// height of the panel
g_panelHeight :LREAL := 0.009;

END_VAR

// ---- GVLs/SlaveArms/GVL_SlaveControlParameters.TcGVL
{attribute 'global_init_slot' := '49991'}
VAR_GLOBAL CONSTANT
	// slave arm joint position controller parameters
	g_posKp :ARRAY[1..g_sJntNum] OF LREAL :=[2000.0, 2000.0, 18000.0, 5(5)];
	g_posKd :ARRAY[1..g_sJntNum] OF LREAL :=[200.0, 200.0, 1800.0, 5(0.25)];
	g_posKi :ARRAY[1..g_sJntNum] OF LREAL :=[20000.0, 20000.0, 30000.0, 5(10.0)];
	g_posKiLimit :ARRAY[1..g_sJntNum] OF LREAL :=[2500,2500,  250, 5(75)];// define in current
	g_posCtrlLimit :ARRAY[1..g_sJntNum] OF LREAL :=[5600,5600,  500, 5(200)];// define in current
	
	// slave arm joint position controller parameters-----Modify joint stiffness---More flexible--1028
	g_allowLowStiff:BOOL:=FALSE;
	g_posKpLowStiff :ARRAY[1..g_sJntNum] OF LREAL :=[500.0, 500.0, 18000.0, 5(5)];
	g_posKdLowStiff :ARRAY[1..g_sJntNum] OF LREAL :=[200.0, 200.0, 1800.0, 5(0.25)];
	g_posKiLowStiff :ARRAY[1..g_sJntNum] OF LREAL :=[10000.0, 10000.0, 30000.0, 5(10.0)];
	g_posKiLimitLowStiff :ARRAY[1..g_sJntNum] OF LREAL :=[500,1000,  250, 5(75)];// define in current
	g_posCtrlLimitLowStiff :ARRAY[1..g_sJntNum] OF LREAL :=[500,1000,  500, 5(250)];// define in current
	
	// control tolerance
	g_jntCtrlAngTolLow :LREAL :=0.2*g_deg2Rad;
	g_jntCtrlAngTolHigh :LREAL :=2*g_deg2Rad;
	g_cartCtrlPosTolLow :LREAL :=0.0002;
	g_cartCtrlOriTolLow :LREAL :=0.2*g_deg2Rad;
	g_cartCtrlPosTolHigh :LREAL :=0.001;
	g_cartCtrlOriTolHigh :LREAL :=2*g_deg2Rad;
	
	// filter cut-off frequency for velocity and torque
	g_curJntVelLpfCutoffFreq :LREAL := 30;
	g_cmdJntTrqLpfCutoffFreq :LREAL := 300;
	g_curJntTrqLpfCutoffFreq :LREAL := 300;
		
	// controller would keep command unchanged when error 
	// between command and current value is less than this value
	g_jntCtrlErrForCmdHold :LREAL :=1.0*g_deg2Rad;
	
	// joint is assumed to be static if velocity is less than this value
	g_jntStaticVelThres :LREAL :=0.2*g_deg2Rad;
	
	// joint velocity threshold for full friction compensation
	g_fullFrictionVel :LREAL :=2.0*g_deg2Rad;
	
	// friciton compensation scael
	g_frictionCompScale :LREAL := 0.8;
	
END_VAR

// ---- GVLs/SlaveArms/GVL_SlaveJointEncoderCaliData.TcGVL
{attribute 'qualified_only'}
// Robot3 --joints parameters of slave arms
VAR_GLOBAL CONSTANT	
	// absolute encoder value at minimal joint positon
	g_minLinkEncoder :ARRAY[1..g_sArmNum, 1..g_sJntNum] OF DINT :=
		[796618, 12395160, 5368016, 0, 0, 0, 0, 0,
		 13317378, 3888760, 9175760, 0, 0, 0, 0, 0,
		 823964, 3955316, 15205696, 0, 0, 0, 0, 0,
		 4820816, 7977020, 9226720, 0, 0, 0, 0, 0];
		 
	// absolute encoder value at maximum joint positon
	g_maxLinkEncoder :ARRAY[1..g_sArmNum, 1..g_sJntNum] OF DINT :=
		[15464922, 5123844, 14570432, 0, 0, 0, 0, 0,
		 11230582, 13464106, 1613344, 0, 0, 0, 0, 0,
		 15526052, 13536910, 7701984, 0, 0, 0, 0, 0,
		 2731020, 789080, 1671808, 0, 0, 0, 0, 0];
	
	// absolute encoder value at calibrated positon
	g_caliLinkEncoder :ARRAY[1..g_sArmNum, 1..g_sJntNum] OF DINT :=
		[8162412, 8169482, 14570432, 15377856,15482848, 7058832, 7015248, 7155184,
		 3932766, 16656494, 1613344, 15324752, 15485488, 7135776, 7032592, 6946704,
		 8248074, 16595424, 7701984, 15349408, 15361392, 7017904, 6757296, 7028608,
		 12196142, 3807946, 1671808, 15274368, 15387696, 6812992, 7016768, 7073088];
	
	 // if absolute encoder value cross zeros within joint motion range
	 // NOTICE: joint 7 is always 0.
	g_linkEncZeroCross :ARRAY[1..g_sArmNum, 1..g_sJntNum] OF INT :=
		[0, 0, 0, 1, 1, 1, 1, 1,
		 1, 1, 1, 1, 1, 1, 1, 1,
		 0, 1, 1, 1, 1, 1, 1, 1,
		 1, 0, 1, 1, 1, 1, 1, 1];
		 
	 // joint SDO address
	g_slaveArmNetID: ARRAY[1..4] OF T_AmsNetId:=['169.254.186.39.3.1','169.254.186.39.8.1','169.254.186.39.9.1','169.254.186.39.10.1'];
	g_slaveJointNetPort:ARRAY[1..g_sArmNum,1..g_sJntNum] OF UINT :=[
		1006,	1007,	1008,	2(1009),	3(1010),
		1006,	1007,	1008,	2(1009),	3(1010),
		1006,	1007,	1008,	2(1009),	3(1010),
		1006,	1007,	1008,	2(1009),	3(1010)];
	g_slaveLEDNetPort:ARRAY[1..g_sArmNum] OF UINT :=[4(1004)];
		
//################ DO NOT modify parameters below ###########################
	// abolute encoder expanded limit buffer in case there is calibrtion error at limit position
	g_linkEncLimitBuffer : DINT := 100000;
	
	// absolute encoder direction
	g_asbEncoderDir :ARRAY[1..g_sJntNum] OF INT :=[1, -1, 1, 1, 1, 1, 1, 1];
	
	// flag if joint can rotate multiple cycles
	g_multipleCyclesJoint :ARRAY[1..g_sArmNum, 1..g_sJntNum] OF INT :=
		[0, 0, 0, 1, 1, 1, 1, 1,
		 0, 0, 0, 1, 1, 1, 1, 1,
		 0, 0, 0, 1, 1, 1, 1, 1,
		 0, 0, 0, 1, 1, 1, 1, 1];
		 
	// joint position at link encoder calibrated point
	g_linkEncCaliJntPos :ARRAY[1..g_sJntNum] OF LREAL :=[0.0, -PI/2 + 8*g_deg2rad, 0.581633, 5(0.0)];

	
END_VAR

// ---- GVLs/SlaveArms/GVL_SlaveMotorParameters.TcGVL
{attribute 'global_init_slot' := '49991'}
{attribute 'qualified_only'}
VAR_GLOBAL CONSTANT
	// encoder resolution
	g_incEncoderRes :ARRAY[1..g_sJntNum] OF DINT :=[8(65536)];
	g_absEncoderRes :ARRAY[1..g_sJntNum] OF DINT :=[8(16777216)];
	
	// reduction ratio
	g_motorReduction :ARRAY[1..g_sJntNum] OF LREAL :=[ 81,81,  (66.0/10)*2*pi/0.010, 5(388125.0/4693)];
	g_absEncoderReduction :ARRAY[1..g_sJntNum] OF LREAL :=[2(1.0), 2*PI/0.64, 5(1.0)];
	
	// motor parameters
	g_motorTrqConst :ARRAY[1..g_sJntNum] OF LREAL :=[ 0.16,0.16, 0.017,5(0.0193)];
	g_motorMaxCurrent :ARRAY[1..g_sJntNum] OF LREAL :=[ 5600,5600,  600, 5(250)];//mA
	
	// motor encoder direction
	g_motorDir :ARRAY[1..g_sJntNum] OF INT :=[-1, 1, -1, 1, 1, 1, 1, 1];
																 
	// joint position limit
	g_minJntPos: ARRAY[1..g_sJntNum] OF LREAL:=[-2.7,	-1.5-pi/2,	0.23, 	5(-g_largeNum)];	
	g_maxJntPos: ARRAY[1..g_sJntNum] OF LREAL:=[2.7,	1.13-pi/2, 	0.58, 		5(g_largeNum)];
	
	// DH joint position limit
	//NOTE: wrist pitch and yaw angle is reset after instrument is mounted 
	g_minDHJntPos : ARRAY[1..6] OF LREAL :=[-2.7,	-1.2-pi/2,	0.235, -5.5, -PI/2 - 75*g_deg2Rad , -PI/2];
	g_maxDHJntPos : ARRAY[1..6] OF LREAL :=[2.7,	1-pi/2, 	0.575, 5.5, -PI/2 + 75*g_deg2Rad, PI/2];
	
	// joint velocity limit
	g_maxJntVel :ARRAY[1..g_sJntNum] OF LREAL :=[1.25, 1.25, 0.25, 5(7.0)];
		
END_VAR

// ---- FBs_CartControlles/I_CartJointCtrl.TcIO
INTERFACE I_CartJointCtrl

METHOD init : BOOL
VAR_IN_OUT CONSTANT
	i_slaveCart	:FB_SlaveCart;
END_VAR
VAR_IN_OUT 
	r_cartCtrlCmd :ST_SlaveArmCtrlCmds;
END_VAR
END_METHOD

PROPERTY isFinished : BOOL
GET
END_GET
END_PROPERTY

METHOD reset : BOOL
VAR_INPUT
END_VAR
END_METHOD

METHOD run : BOOL
VAR_IN_OUT CONSTANT
	i_slaveCart	:FB_SlaveCart;
END_VAR
VAR_IN_OUT 
	r_cartCtrlCmd :ST_SlaveArmCtrlCmds;
END_VAR
END_METHOD

END_INTERFACE

// ---- FBs_SlaveControllers/I_SlaveArmCtrl.TcIO
INTERFACE I_SlaveArmCtrl

METHOD init : BOOL
VAR_IN_OUT CONSTANT
	i_slaveArm	:FB_SlaveArm;
END_VAR
VAR_IN_OUT 
	r_slaveArmCtrlCmd :ST_SlaveArmCtrlCmds;
END_VAR
END_METHOD

PROPERTY isFinished : bool
GET
END_GET
END_PROPERTY

METHOD reset : BOOL
VAR_INPUT
END_VAR
END_METHOD

METHOD run : BOOL

VAR_IN_OUT CONSTANT
	i_endoscopePose : ST_Frame;
	i_masterStatus :ST_MasterStatus;
	i_setupStatus: ST_SetupStatus;
	i_slaveArm :FB_SlaveArm;
	
END_VAR
VAR_IN_OUT
	r_slaveArmCtrlCmd :ST_SlaveArmCtrlCmds;
END_VAR
END_METHOD

PROPERTY timePeriod : lreal
GET
END_GET
END_PROPERTY

END_INTERFACE

// ---- Mains/CartControl.TcPOU
PROGRAM CartControl
VAR
	// cart instance
	m_cartRobot :FB_CartRobot;
	
	// Output cart status
	m_cartStatus AT%Q* : ST_CartStatus;
	
	// cart joint data
	m_cartJointsData AT %Q* :ST_CartJointData;
	
	m_cartDataPool: ST_CartInputDataPool;
	
	// wait time before cart init for ethercat to be statble 
	m_cartInitWaitTime : LREAL:=0;
	
	// cart init flag
	m_cartInit :BOOL :=FALSE;
	
	m_workHeartTon0 : TON;
	m_workHeartTon1 : TON;
	
	m_cartInSterileStateTon :Ton;
	m_cartInSterileState :BOOL;
	//Aseptic sleeve is installed flag
	m_asepticInstalledFlag : Vec4b;
	m_slaveArmDisableFlag : Vec4b;
END_VAR

// wait communication to be stable
IF(m_cartInitWaitTime<g_robotInitWaitTime) THEN
	m_cartInitWaitTime := m_cartInitWaitTime+g_cartCtrlCycleTime;
	RETURN;
END_IF

// cart init
IF m_cartInit =FALSE THEN
	m_cartRobot.Init();
	m_cartInit:=TRUE;
END_IF

// input from UI
UIInputProcess();

// cart run
m_cartRobot.run(m_cartDataPool);

m_cartRobot.getStatus(m_cartStatus,m_cartJointsData);


UIOutputProcess();

// tranform data from UI(global variable write by ADS) to ST_UIData
METHOD UIInputProcess : BOOL
VAR_INPUT
END_VAR
VAR
	i:int;
END_VAR
// cart Joystick data
m_cartDataPool.m_UIData.m_joystickDataFromUI := GVL_interactUI.g_joystickSignalArray;

m_cartDataPool.m_UIData.m_ctrlEnableFromUI := GVL_interactUI.g_uiCtrl;

//limit_height:UINT;  上位机的高度值单位是mm，系统的高度值单位是m，底座高度是1805mm
//打开ui_control.limit_height_adjusting后可以调整立柱，并实时将立柱当前高度上传
IF (GVL_interactUI.g_uiCtrl.m_heightLimitAdjustEnable=TRUE) THEN
	m_cartDataPool.m_UIData.m_standColumnHightLimit := GVL_CartMotorParameters.g_maxJntPos[5];
ELSIF  (GVL_interactUI.g_uiCtrl.m_heightLimitAdjustEnable=FALSE) AND GVL_interactUI.g_heightLimitEnbale AND ABS((m_cartDataPool.m_UIData.m_standColumnHightLimit *1000+1850)-GVL_interactUI.g_heightLimitFromUI)>5 THEN
	m_cartDataPool.m_UIData.m_standColumnHightLimit := UINT_TO_LREAL(GVL_interactUI.g_heightLimitFromUI-GVL_CartControlParameters.g_cartInitialHeight)/1000;
ELSIF GVL_interactUI.g_heightLimitEnbale=FALSE THEN
	m_cartDataPool.m_UIData.m_standColumnHightLimit := GVL_CartMotorParameters.g_maxJntPos[5];
END_IF
GVL_interactUI.g_heightLimit :=LREAL_TO_UINT (m_cartRobot.m_slaveCart.curJntPos[5] * 1000 + GVL_CartControlParameters.g_cartInitialHeight);

//Surgical orientation selection
m_cartDataPool.m_UIData.m_surgicalSite := GVL_interactUI.g_surgicalSite;
m_cartDataPool.m_UIData.m_surgicalLocation := GVL_interactUI.g_surgicalLocation;
END_METHOD

METHOD UIOutputProcess : BOOL
VAR_INPUT
END_VAR
VAR 
	i : INT;
END_VAR
//TODO
//work heart
m_workHeartTon0(IN:= GVL_interactUI.g_heartBeat = 1, PT:= T#1S, Q=> , ET=> );
m_workHeartTon1(IN:= GVL_interactUI.g_heartBeat = 0, PT:= T#1S, Q=> , ET=> );
IF m_workHeartTon0.Q THEN
	GVL_interactUI.g_heartBeat :=0 ;
ELSIF m_workHeartTon1.Q THEN
	GVL_interactUI.g_heartBeat  :=1 ;
END_IF

GVL_interactUI.g_cartOperation.m_drapingAdjustState := m_cartRobot.m_slaveCart.m_cartDataFromUI.m_cartDrapingState;
GVL_interactUI.g_cartOperation.m_dockingAdjustState := m_cartRobot.m_slaveCart.m_cartDataFromUI.m_cartDockingState;

GVL_interactUI.g_trocarStatus := INT_TO_BOOL(m_cartRobot.m_slaveCart.m_trocarOnFlag);

GVL_interactUI.g_slaveRunAlone := NOT SlaveArmControl.m_slaveRobot.m_masterOnLine;
GVL_interactUI.g_joysticksTrigger := SafetyCheck.m_joysticksTrigger;

IF GVL_interactUI.g_surgicalStatus = 1 THEN
	IF NOT SlaveArmControl.m_slaveRobotData.m_asepticDeployCompletedFlag THEN
		m_slaveArmDisableFlag := g_zeroVec4b;
	END_IF
	GVL_interactUI.g_cartOperation.m_setupSterileState := BOOL_TO_UINT(m_asepticInstalledFlag[1]) OR BOOL_TO_UINT(m_asepticInstalledFlag[2]) OR BOOL_TO_UINT(m_asepticInstalledFlag[3]) OR BOOL_TO_UINT(m_asepticInstalledFlag[4]) ;
ELSE
	GVL_interactUI.g_cartOperation.m_setupSterileState := BOOL_TO_UINT(m_asepticInstalledFlag[1]) AND BOOL_TO_UINT(m_asepticInstalledFlag[2]) AND BOOL_TO_UINT(m_asepticInstalledFlag[3]) AND BOOL_TO_UINT(m_asepticInstalledFlag[4]) ;
	m_slaveArmDisableFlag := SlaveArmControl.m_slaveInputDataPool.m_UIData.m_slaveArmDisableFlag;	
	Gvl_interactUI.g_InstruSeriesRecord := g_zeroInstruRecord;
END_IF

FOR i := 1 TO 4 BY 1 DO
	m_asepticInstalledFlag[i] := m_slaveArmDisableFlag[i] OR SlaveArmControl.m_slaveRobot.m_panelMountedFlag[i];
END_FOR

GVL_interactUI.g_cartOperation.m_setupSterileStateArm1 := BOOL_TO_UINT(m_asepticInstalledFlag[1]); 
GVL_interactUI.g_cartOperation.m_setupSterileStateArm2 := BOOL_TO_UINT(m_asepticInstalledFlag[2]); 
GVL_interactUI.g_cartOperation.m_setupSterileStateArm3 := BOOL_TO_UINT(m_asepticInstalledFlag[3]); 
GVL_interactUI.g_cartOperation.m_setupSterileStateArm4 := BOOL_TO_UINT(m_asepticInstalledFlag[4]); 

GVL_interactUI.g_cartOperation.m_scopeInstalled := BOOL_TO_UINT(m_cartDataPool.m_slaveStatus.m_endoscopeMounted);

FOR i := 1 TO 4 BY 1 DO
	IF SlaveArmControl.m_slaveRobot.m_slaveArms[i].instrument.Instrutype<>InstruType_endoscope THEN
		IF SlaveArmControl.m_slaveRobot.m_instrumentMountedFlag[i] AND SlaveArmControl.m_slaveRobot.m_endoscopeMounted AND GVL_interactUI.g_cartOperation.m_setupSterileState = 1 THEN
			GVL_interactUI.g_cartOperation.m_inSurgicalAllowed := 1;
			EXIT;
		ELSE
			GVL_interactUI.g_cartOperation.m_inSurgicalAllowed := 0;
		END_IF	
	END_IF	
END_FOR


//Cart_static_in_sterile_state:UINT; //台车进入无菌区，并且台车停止运动(连续10s没有运动)，0：没有完成，1：完成
IF m_cartRobot.m_slaveCart.m_cartDataFromUI.m_cartDockingState = 1 THEN
	IF m_cartRobot.m_CartState = CartJointState_Movement THEN
		m_cartInSterileState := FALSE;
	ELSIF m_cartRobot.m_lastCartState = CartJointState_Movement THEN
		m_cartInSterileState := TRUE;
	END_IF
ELSE
	m_cartInSterileState := FALSE;
	GVL_interactUI.g_cartOperation.m_cartInSterileState:=0;
END_IF
m_cartInSterileStateTon(IN:= m_cartInSterileState, PT:= T#10S, Q=> , ET=> );
IF m_cartInSterileStateTon.Q THEN
	GVL_interactUI.g_cartOperation.m_cartInSterileState:=1;
END_IF
END_METHOD

END_PROGRAM

// ---- FBs_Robots/FB_CartRobot.TcPOU
FUNCTION_BLOCK FB_CartRobot
VAR_INPUT
END_VAR
VAR_OUTPUT
END_VAR
VAR

	m_slaveCart: FB_SlaveCart;		
	
	// input arm button 
	m_carHandChassisDriveUnlock AT%I* :ARRAY [1..2] OF BOOL;
	
	//open laser io
	m_openHorizonLaser AT  %Q* :DINT;
	m_openCrossLaser AT  %Q* :DINT;

	m_joystickData:Vec8d;

	// all cart controller instance 
	m_cartCtrlFactory :ARRAY[1..CartJointState_totalNum] OF I_CartJointCtrl;
	
	m_cartState:E_CartJointState:=CartJointState_Init;
	m_lastCartState:E_CartJointState:=CartJointState_Init;
	m_nextCartState:E_CartJointState:=CartJointState_Init;
	
	// flag if cart joint self-check passed
	m_selfCheckPass:  BOOL :=FALSE;
	
	// all cart controller instance 
	m_cartError :FB_CartCtrlError;
	m_cartInit :FB_CartCtrlInit;
	m_cartReady :FB_CartCtrlReady;
	m_cartInSurgery :FB_CartCtrlInSurgery;
	m_cartMotionCar :FB_CartCtrlMotionCar;
	m_cartAsepticDeploy :FB_CartCtrlAsepticDeploy;
	m_cartAdjust :FB_CartCtrlAdjust;
	m_cartRotaOverhang :FB_CartCtrlRotaOverhang;
	m_cartSlowStop : FB_CartCtrlSlowDown;
	m_cartStandColuAdjust : FB_CartCtrlStandColuAdjust;
	
	// cart controller interface
	m_cartCtrl : I_CartJointCtrl;
	m_cartCtrlCmds : ST_SlaveArmCtrlCmds;
	
	//state machine flow jump condition allowed
	m_hangAdjustAllowed : BOOL;
	m_asepticDeploymentAllowed :BOOL;
	m_cartMoveAllowed :BOOL;
	m_rotaOverhangAllowed :BOOL;
END_VAR

METHOD getStatus : BOOL
VAR_IN_OUT
	
	r_cartStatus :ST_CartStatus;	

	// cart joint data
	r_cartJointsData :ST_CartJointData;
END_VAR

VAR 
	i : INT;
END_VAR
r_cartStatus.m_CartState :=m_cartState;

r_cartStatus.m_uiControl := GVL_interactUI.g_uiCtrl;
r_cartStatus.m_cartDumpEnergy := GVL_interactUI.g_dumpEnergyUPS;
r_cartStatus.m_sdrivingLeverSensorManualFlag :=NOT m_slaveCart.m_drivingLeverSensorManual;
//r_cartStatus.m_stabilizerDeployedFlag
r_cartStatus.m_trocarOnFlag := m_slaveCart.m_trocarOnFlag;
r_cartStatus.m_joystickValue := m_slaveCart.m_joystickSignal;
r_cartStatus.m_jntPosReachLimit := m_cartAdjust.jntPosReachLimit;

r_cartJointsData.m_cmdJntPos := m_slaveCart.cmdJntPos;
r_cartJointsData.m_cmdJntVel := m_slaveCart.cmdJntVel;
r_cartJointsData.m_curJntPos := m_slaveCart.curJntPos;
r_cartJointsData.m_curJntTrq := m_slaveCart.curJntCurrent;
r_cartJointsData.m_curJntVel := m_slaveCart.curJntVel;
r_cartJointsData.m_curLinkPos := m_slaveCart.curLinkPos;
r_cartJointsData.m_curMotorPos := m_slaveCart.curMotorPos;
END_METHOD

METHOD init : BOOL
VAR_INPUT
END_VAR
VAR
	i:INT;
END_VAR

m_slaveCart.init();
m_cartState := CartJointState_Init;
m_lastCartState := CartJointState_Init;
m_nextCartState := CartJointState_Init;
m_selfCheckPass := FALSE;

//command init
m_cartCtrlCmds.m_jntEnableFlag := g_zeroVec8i;
m_cartCtrlCmds.m_jntOPMode := g_slaveAllPosMode;
m_cartCtrlCmds.m_cmdJntPos := m_slaveCart.m_curJntPos;
m_cartCtrlCmds.m_cmdJntVel := g_zeroVec8d;
m_cartCtrlCmds.m_cmdJntAcc := g_zeroVec8d;
m_cartCtrlCmds.m_cmdJntTrq := g_zeroVec8d;


// generate controller factory
//m_cartCtrlFactory[CartJointState_Error] := m_cartError;
m_cartCtrlFactory[CartJointState_Init] := m_cartInit;
m_cartCtrlFactory[CartJointState_Ready] := m_cartReady;
m_cartCtrlFactory[CartJointState_InSurgery] := m_cartInSurgery;
m_cartCtrlFactory[CartJointState_Movement] := m_cartMotionCar;
m_cartCtrlFactory[CartJointState_HangAdjust] := m_cartAdjust;
m_cartCtrlFactory[CartJointState_AsepticDeployment] := m_cartAsepticDeploy;
m_cartCtrlFactory[CartJointState_RotaOverhang] := m_cartRotaOverhang;
m_cartCtrlFactory[CartJointState_SlowStop] := m_cartSlowStop;
m_cartCtrlFactory[CartJointState_StandColuAdjust] := m_cartStandColuAdjust;

// assign controller
m_cartCtrl:=m_cartCtrlFactory[m_cartState];
m_cartCtrl.Init(m_slaveCart,m_cartCtrlCmds);
END_METHOD

METHOD laserIO : BOOL
VAR_INPUT
END_VAR

//cross laser IO output , when slave self check succeed , and trocar  install at least one
IF GVL_interactUI.g_slaveSelfCheckStatus = 2 AND m_slaveCart.m_trocarOnFlag = 0 THEN
	m_openCrossLaser := 1;
ELSE
	m_openCrossLaser := 0;
END_IF

//Horizontal laser IO output ,when adjusting the trolley or moving the trolley
IF (m_slaveCart.curJntPos[5] * 1000 + GVL_CartControlParameters.g_cartInitialHeight) > GVL_CartControlParameters.g_cartOpenHorizonLaserHeight AND  (m_cartState = CartJointState_Movement OR m_cartState = CartJointState_HangAdjust) THEN
	m_openHorizonLaser :=  1;
ELSE
	m_openHorizonLaser :=  0;
END_IF
END_METHOD

METHOD PUBLIC run : BOOL
VAR_IN_OUT CONSTANT
	i_cartDataPool: ST_CartInputDataPool;
END_VAR
VAR
	i:INT;
END_VAR
// state machine transition
stateMachine(i_cartDataPool);	

//update ui data
m_slaveCart.ProcessingUIData(i_cartDataPool.m_UIData);

//update cart joint status
m_slaveCart.updateStatus();

laserIO();

// null ptr check
IF 0 = m_cartCtrl THEN
	RETURN;
END_IF

// run controller
m_cartCtrl.run(m_slaveCart,m_cartCtrlCmds);


m_slaveCart.updateCmds(m_cartCtrlCmds);
END_METHOD

METHOD PROTECTED stateMachine : BOOL
VAR_IN_OUT CONSTANT
	i_cartDataPool: ST_CartInputDataPool;
END_VAR
VAR
	i,j:INT;
END_VAR
m_hangAdjustAllowed := m_slaveCart.m_trocarOnFlag=0 AND ( i_cartDataPool.m_UIData.m_ctrlEnableFromUI.m_joystickEnable OR i_cartDataPool.m_UIData.m_ctrlEnableFromUI.m_cameraJoystickEnable);
m_asepticDeploymentAllowed := m_slaveCart.m_trocarOnFlag=0 AND ((i_cartDataPool.m_UIData.m_ctrlEnableFromUI.m_dockingEnable AND m_slaveCart.cartDockingState=0) 
												OR (i_cartDataPool.m_UIData.m_ctrlEnableFromUI.m_drapingEnable AND m_slaveCart.cartDrapingState=0)) AND NOT ( i_cartDataPool.m_safetyData.m_cartAdjustErr OR i_cartDataPool.m_safetyData.m_cartStandColumnErr) ;
m_cartMoveAllowed := m_slaveCart.m_trocarOnFlag=0 AND  m_carHandChassisDriveUnlock[1] AND m_carHandChassisDriveUnlock[2] AND NOT i_cartDataPool.m_safetyData.m_cartWheelErr;
m_rotaOverhangAllowed := m_slaveCart.m_trocarOnFlag=0 AND m_slaveCart.m_rotaOverhangOnFlag > 0 AND NOT i_cartDataPool.m_safetyData.m_cartOverhangErr;

// state machine transit
CASE m_cartState OF
	//cart joint error
	CartJointState_Error:
		//IF FALSE = i_cartDataPool.m_safetyData.m_slaveErrFlag THEN
		//	// to standby
		//	IF m_selfCheckPass THEN
		//		m_nextCartState :=CartJointState_Standby;
		//	ELSE
		//		m_nextCartState :=CartJointState_Init;
		//	END_IF
		//END_IF

	CartJointState_Init:
		IF m_cartCtrl.isFinished THEN
			m_nextCartState :=CartJointState_Ready;
		END_IF
		
		
	CartJointState_Ready:
		IF m_cartCtrl.isFinished  THEN
			m_nextCartState := CartJointState_InSurgery;
			
		ELSIF m_hangAdjustAllowed THEN
			m_nextCartState := CartJointState_HangAdjust;
			
		ELSIF m_asepticDeploymentAllowed THEN
			m_nextCartState := CartJointState_AsepticDeployment;
			
		ELSIF m_cartMoveAllowed THEN
			m_nextCartState := CartJointState_Movement;
			
		ELSIF m_rotaOverhangAllowed THEN
			m_nextCartState := CartJointState_RotaOverhang;
			
		ELSIF m_slaveCart.m_trocarOnFlag=0 AND  m_slaveCart.m_columnAdjustEnable  THEN
			m_nextCartState := CartJointState_StandColuAdjust;
		END_IF
		
	
	CartJointState_InSurgery:
		IF m_cartCtrl.isFinished  THEN
			m_nextCartState :=CartJointState_Ready;
		END_IF
		
		
	CartJointState_Movement:
		IF m_slaveCart.m_trocarOnFlag<>0 OR (NOT m_carHandChassisDriveUnlock[1] AND NOT m_carHandChassisDriveUnlock[2])  THEN
			m_nextCartState :=CartJointState_Ready;
		ELSIF i_cartDataPool.m_safetyData.m_cartWheelErr THEN
			m_nextCartState :=CartJointState_Ready;
		END_IF
		
		
	CartJointState_HangAdjust:
		IF  m_slaveCart.m_trocarOnFlag<>0 OR (NOT i_cartDataPool.m_UIData.m_ctrlEnableFromUI.m_joystickEnable AND NOT i_cartDataPool.m_UIData.m_ctrlEnableFromUI.m_cameraJoystickEnable ) THEN
			m_nextCartState :=CartJointState_SlowStop;
		END_IF
		
		
	CartJointState_AsepticDeployment:
		IF m_cartCtrl.isFinished  THEN
			IF i_cartDataPool.m_UIData.m_ctrlEnableFromUI.m_dockingEnable THEN
				m_slaveCart.cartDockingState := 1;
			ELSIF i_cartDataPool.m_UIData.m_ctrlEnableFromUI.m_drapingEnable THEN
				m_slaveCart.cartDrapingState := 1;
			END_IF
			m_nextCartState :=CartJointState_SlowStop;
		ELSIF i_cartDataPool.m_safetyData.m_cartAdjustErr OR i_cartDataPool.m_safetyData.m_cartStandColumnErr THEN
			m_nextCartState :=CartJointState_Ready;
		ELSIF m_slaveCart.m_trocarOnFlag<>0 OR (NOT i_cartDataPool.m_UIData.m_ctrlEnableFromUI.m_dockingEnable AND NOT i_cartDataPool.m_UIData.m_ctrlEnableFromUI.m_drapingEnable) THEN
			m_nextCartState :=CartJointState_SlowStop;
		END_IF
		
		
	CartJointState_RotaOverhang:
		IF m_slaveCart.m_rotaOverhangOnFlag = 0 OR  m_slaveCart.m_trocarOnFlag<>0  THEN
			m_nextCartState :=CartJointState_SlowStop;
		ELSIF i_cartDataPool.m_safetyData.m_cartOverhangErr THEN
			m_nextCartState :=CartJointState_Ready;
		END_IF
		
	CartJointState_StandColuAdjust:
		IF (m_slaveCart.m_trocarOnFlag<>0 OR i_cartDataPool.m_safetyData.m_cartStandColumnErr) OR  NOT m_slaveCart.m_columnAdjustEnable  THEN
			m_nextCartState :=CartJointState_SlowStop;
		END_IF	
	
	CartJointState_SlowStop:
		IF m_cartCtrl.isFinished  THEN
			m_nextCartState :=CartJointState_Ready;
		END_IF
END_CASE

// Controller transit
IF m_nextCartState<> m_cartState THEN
	//reset current controller
	m_cartCtrl.reset();
	
	// transit to new controller
	m_lastCartState:=m_cartState;
	m_cartState:=m_nextCartState;
	m_cartCtrl:=m_cartCtrlFactory[m_cartState];
	
	//init next controller
	m_cartCtrl.Init(m_slaveCart, m_cartCtrlCmds);
	m_slaveCart.updateCmds(m_cartCtrlCmds);
END_IF
END_METHOD

END_FUNCTION_BLOCK

// ---- FBs_Robots/FB_SlaveCart.TcPOU
FUNCTION_BLOCK FB_SlaveCart
VAR
	
	//Driving force of the car io
	m_driveForce AT %I* :Vec2i;
	
	//stabilizing foot sensor  (normally-closed contact)
	m_stabilizFootSensorLeft AT%I* :BOOL;
	m_stabilizFootSensorRight AT%I* :BOOL;
	m_drivingLeverSensorAuto AT%I* :BOOL;
	m_drivingLeverSensorManual AT%I* :BOOL;
	
	//Trocar IO check
	m_trocarIO AT %I* : ARRAY [1..4] OF UDINT;
	m_trocarCheck : ARRAY [1..4] OF FB_trocarDetect;
	m_trocarFlag : ARRAY [1..4] OF BOOL;
	m_trocarOnFlag : INT:=0;
	
	//output screw break IO 
	m_screwBreak AT %Q* : BOOL;
	m_screwBreakSR : SR;
	
	//car overhang rotation signal is in the arm
	m_carRotaOverhangIO AT%I* : ARRAY [1..4] OF UDINT;
	m_rotaButtonDetect : ARRAY [1..4] OF FB_rotaButtonDetect;
	m_rotaOverhangOnFlag : UDINT :=0;
	
	//cart joint
	m_cartJoints: ARRAY [1..g_cartJntNum] OF FB_CartJoint;
	
	// cart status
	m_cartStatus  : ST_CartStatus;
	
	//cart joint 5 enable detect
	m_standColumnEnableDetect : FB_cartJntEnableDetect;
	m_standColumnDisenableDetect : FB_cartJntDisenableDetect;

	// arm joint data
	m_curMotorPos :Vec8d;
	m_curLinkPos :Vec8d;
	m_curLinkSingle :Vec8d;
	m_curJntPos :Vec8d;
	m_curDHJntPos :Vec6d;
	m_curGripAngle :LREAL;
	m_curJntVel :Vec8d;
	m_curDHJntVel :Vec6d;
	m_curJntTrq :Vec8d;
	m_rawJntCurrent :Vec8d;
	m_filtJntCurrent :Vec8d;
	m_cmdJntTrq :Vec8d;
	m_cmdJntCurrent : Vec8d;
	m_cmdJntPos :Vec8d;
	m_cmdJntVel :Vec8d;

	//SDO Writer
	m_CommunicationCycleInitMZSub1:ARRAY [1..3] OF FB_EcCoESdoWrite;
	m_CommunicationCycleInitMZSub2:ARRAY [1..3] OF FB_EcCoESdoWrite;
	m_CommunicationCycleSub1:INT:=1;
	m_CommunicationCycleSub2:INT:=-3;
	
	//update ui information
	m_joystickSignal:Vec8d;
	m_cartDataFromUI : ST_CartUIData;
	m_ctrlEnable : ST_uiControl;
	m_surgicalStatusF : F_TRIG;
	
	//stand column adjust of setup joint 3
	m_columnJntVel : LREAL;
	m_columnAdjustEnable : BOOL;
	m_limitBufferForCtrl : LREAL := 0.01;
	m_midJntPos : LREAL := 0.1;
	enableTon : ARRAY [1..4] OF FB_TON;
	
	// collision detection
	m_collisionDetection : FB_CartCollisionDetect;
	m_collisionFlag :BOOL:=false;
END_VAR

PROPERTY cartDockingState : UINT
GET
END_GET
SET
m_cartDataFromUI.m_cartDockingState := cartDockingState;
END_SET
END_PROPERTY

PROPERTY cartDrapingState : UINT
GET
END_GET
SET
m_cartDataFromUI.m_cartDrapingState := cartDrapingState;
END_SET
END_PROPERTY

METHOD checkIO : BOOL
VAR_INPUT
END_VAR
VAR
	i:INT;
END_VAR
//check overhang rotation button
m_rotaOverhangOnFlag := MAX( m_rotaButtonDetect[1].run(m_carRotaOverhangIO[1]), m_rotaButtonDetect[2].run(m_carRotaOverhangIO[2]),m_rotaButtonDetect[3].run(m_carRotaOverhangIO[3]),m_rotaButtonDetect[4].run(m_carRotaOverhangIO[4]));

FOR i := 1 TO g_sArmNum BY 1 DO
	//trocar in place monitor
	m_trocarFlag[i] := m_trocarCheck[i].run(m_trocarIO[i] );
END_FOR

m_trocarOnFlag := BOOL_TO_INT(m_trocarFlag[1]) + BOOL_TO_INT(m_trocarFlag[2]) + BOOL_TO_INT(m_trocarFlag[3]) + BOOL_TO_INT(m_trocarFlag[4]);

//setup robot joint 3 adjust and drive column movement
m_columnAdjustEnable :=columnAdjustEnable(o_columnJntVel => m_columnJntVel  );
END_METHOD

PROPERTY cmdJntPos : REFERENCE TO Vec8d
GET
cmdJntPos REF= m_cmdJntPos;
END_GET
END_PROPERTY

PROPERTY cmdJntVel : REFERENCE TO Vec8d
GET
cmdJntVel REF= m_cmdJntVel;
END_GET
END_PROPERTY

METHOD columnAdjustEnable : BOOL
VAR_INPUT
END_VAR

VAR_OUTPUT
	o_columnJntVel : LREAL;
END_VAR

VAR_STAT
	curJntPos : vec4d;
	curJntVel : vec4d;
	columnJntVel : vec4d;
	adjustStartFlag : vec4b;
	m_columnAdjustEnable : vec4b;
END_VAR
VAR
	i : INT;
	armId : INT;
	limitDis : vec4d;
	m_adjustFlag : vec4b;
END_VAR

FOR i := 1 TO g_sArmNum DO
	curJntPos[i] := SetupArmControl.m_setupRobot.m_setupArms[i].m_curJntPos[3];
	curJntVel[i] := SetupArmControl.m_setupRobot.m_setupArms[i].m_curJntVel[3];
	m_adjustFlag[i] := SetupArmControl.m_setupRobot.m_setupArms[i].m_manualAdjustOnFlag AND m_trocarOnFlag=0 AND SetupArmControl.m_setupRobot.m_setupArmState[i] = SetupArmState_ManualAdjust 
									AND NOT SafetyCheck.m_SafetyCheck.m_jntErrFlag[i,0,2] AND NOT SafetyCheck.m_SafetyCheck.m_jntErrFlag[i,0,3] AND NOT SafetyCheck.m_SafetyCheck.m_jntErrFlag[i,3,3] AND NOT SafetyCheck.m_SafetyCheck.m_jntErrFlag[i,2,3] ;
	
	IF m_adjustFlag[i] THEN
		limitDis[i] := MIN(GVL_SetupMotorParameters.g_maxJntPos[i,3] - curJntPos[i], curJntPos[i]-GVL_SetupMotorParameters.g_minJntPos[i,3]);
		IF limitDis[i] < m_limitBufferForCtrl THEN
			adjustStartFlag[i] := TRUE; 
			columnJntVel[i] := sign(m_midJntPos - curJntPos[i]) * GVL_CartControlParameters.g_maxJntVel[5];
		
		ELSIF limitDis[i] >= m_limitBufferForCtrl AND NOT m_columnAdjustEnable[i] THEN
			columnJntVel[i] := 0;
			adjustStartFlag[i] := FALSE;
			
		ELSE
			IF curJntVel[i] <> 0 AND adjustStartFlag[i] THEN
				columnJntVel[i] := -LIMIT(-GVL_CartControlParameters.g_maxJntVel[5], curJntVel[i], GVL_CartControlParameters.g_maxJntVel[5]);
			END_IF
		END_IF
		
		armId := i;
		enableTon[i](IN:= adjustStartFlag[i], PT:= T#3S, Q=> m_columnAdjustEnable[i], ET=> );
		EXIT;
	ELSE
		adjustStartFlag[i] := FALSE;
		columnJntVel[i] := 0;
	END_IF
	enableTon[i](IN:= adjustStartFlag[i], PT:= T#3S, Q=> m_columnAdjustEnable[i], ET=> );
END_FOR

//output stand column joint velocity and start adjust single
IF armId > 0 THEN
	o_columnJntVel := columnJntVel[armId];
END_IF
columnAdjustEnable := m_columnAdjustEnable[1] OR m_columnAdjustEnable[2] OR m_columnAdjustEnable[3] OR m_columnAdjustEnable[4];
END_METHOD

PROPERTY ctrlEnable : REFERENCE TO ST_uiControl
GET
ctrlEnable REF= m_ctrlEnable;
END_GET
SET
END_SET
END_PROPERTY

PROPERTY curDHJntPos :REFERENCE TO Vec6d
GET
curDHJntPos ref= m_curDHJntPos;
END_GET
END_PROPERTY

PROPERTY curDHJntVel :REFERENCE TO Vec6d
GET
curDHJntVel REF= m_curDHJntVel;
END_GET
END_PROPERTY

PROPERTY curJntCurrent :REFERENCE TO Vec8d
GET
curJntCurrent ref=m_filtJntCurrent;
END_GET
END_PROPERTY

PROPERTY curJntPos : REFERENCE TO Vec8d
GET
curJntPos ref=m_curJntPos;
END_GET
END_PROPERTY

PROPERTY curJntVel :REFERENCE TO Vec8d
GET
curJntVel ref=m_curJntVel;
END_GET
END_PROPERTY

PROPERTY curLinkPos :REFERENCE TO Vec8d
GET
curLinkPos ref=m_curLinkPos;
END_GET
END_PROPERTY

PROPERTY curMotorPos : REFERENCE TO  Vec8d
GET
curMotorPos ref=m_curMotorPos;
END_GET
END_PROPERTY

METHOD PUBLIC enable : BOOL
VAR_IN_OUT CONSTANT
	i_jntIdx :Vec8i;
END_VAR
VAR
	i :INT ;
END_VAR
FOR i:=1 TO g_cartJntNum DO
	IF 3<=i AND i<5 THEN
		IF 1= i_jntIdx[i] THEN
			m_cartJoints[i].enableMZ();
		ELSE
			m_cartJoints[i].disable();
		END_IF
	ELSIF i = 5 THEN
		IF 1= i_jntIdx[i] THEN
			m_screwBreak := m_standColumnEnableDetect.run(IOValue:= m_cartJoints[i].enableMZ());
			m_standColumnDisenableDetect.run(IOValue:=FALSE );
		ELSE
			m_standColumnEnableDetect.run(IOValue:= FALSE);
			m_screwBreak :=  NOT m_standColumnDisenableDetect.run(IOValue:=m_cartJoints[i].disable());
		END_IF
	ELSE
		IF 1= i_jntIdx[i] THEN
			m_cartJoints[i].enable();
		ELSE
			m_cartJoints[i].disable();
		END_IF
	END_IF
END_FOR
END_METHOD

METHOD init : BOOL
VAR_INPUT
END_VAR
VAR
	i:INT;
END_VAR


// cart joint init
FOR i:= 1 TO g_cartJntNum BY 1 DO
	m_cartJoints[i].init(i, g_cartCtrlCycleTime);
END_FOR


// joint init
FOR i:=1 TO g_cartJntNum DO
	m_cartJoints[i].initJntPos();
END_FOR


// update cart status if joint position is re-init
updateStatus();



//MingZhi drive example Initialize the communication period
FOR i := 1 TO 3 BY 1 DO
	m_CommunicationCycleInitMZSub1[i](sNetID:= GVL_CartJointEncoderCaliData.g_slaveCartNetID,
				nSlaveAddr := GVL_CartJointEncoderCaliData.g_slaveCartJointNetPort[i+2],
				nSubIndex:=1,nIndex:=16#60C2,pSrcBuf:=ADR(m_CommunicationCycleSub1),cbBufLen:=SIZEOF(m_CommunicationCycleSub1),bExecute:=TRUE);
	
	IF NOT m_CommunicationCycleInitMZSub1[i].bBusy THEN
		m_CommunicationCycleInitMZSub1[i](bExecute:=FALSE);
	END_IF
					
	m_CommunicationCycleInitMZSub2[i](sNetID:= GVL_CartJointEncoderCaliData.g_slaveCartNetID,
					nSlaveAddr := GVL_CartJointEncoderCaliData.g_slaveCartJointNetPort[i+2],
					nSubIndex:=2,nIndex:=16#60C2,pSrcBuf:=ADR(m_CommunicationCycleSub2),cbBufLen:=SIZEOF(m_CommunicationCycleSub2),bExecute:=TRUE);
	
	IF NOT m_CommunicationCycleInitMZSub2[i].bBusy THEN
		m_CommunicationCycleInitMZSub2[i](bExecute:=FALSE);
	END_IF
END_FOR
END_METHOD

METHOD  joystickSignalAnalysis : Vec8d 
VAR_INPUT
	i_joystickDataFromUI:ARRAY [0..21] OF USINT;
END_VAR

VAR_STAT
	i:INT;
	m_handData:ARRAY [0..21] OF USINT;
	m_outHandData : Vec8d;
END_VAR

IF i_joystickDataFromUI[0] = 16#FF THEN
	m_handData := i_joystickDataFromUI;
	m_outHandData[1] :=m_handData[7]*256 + m_handData[8]; // car  joint5 pillar
	m_outHandData[2] :=m_handData[3]*256 + m_handData[4]; //car joint7 beamStretch
	m_outHandData[3] :=m_handData[1]*256 + m_handData[2]; // car joint6  beamRot
	m_outHandData[4] :=m_handData[5]*256 + m_handData[6]; // joint8 overhang 
	m_outHandData[5] :=m_handData[9]*256 + m_handData[10];
	m_outHandData[6] :=m_handData[11]*256 + m_handData[12];
	m_outHandData[7] :=m_handData[13]*256 + m_handData[14];
	m_outHandData[8] :=m_handData[15]*256 + m_handData[16];
END_IF
joystickSignalAnalysis:=m_outHandData;
END_METHOD

METHOD ProcessingUIData : BOOL
VAR_IN_OUT CONSTANT
	//UI information, import from UI controller
	i_UIData :ST_CartUIData;
END_VAR
VAR
	i : INT;
END_VAR
m_joystickSignal := joystickSignalAnalysis(i_UIData.m_joystickDataFromUI);

m_ctrlEnable:=i_UIData.m_ctrlEnableFromUI;

m_cartDataFromUI.m_standColumnHightLimit := i_UIData.m_standColumnHightLimit;

m_cartDataFromUI.m_cartSpecificPosDraping := GVL_CartControlParameters.g_surgicalDrapingPos;

FOR i := 1 TO g_sArmNum BY 1 DO
	IF i_UIData.m_surgicalSite > 0 AND i_UIData.m_surgicalLocation > 0 THEN
		m_cartDataFromUI.m_cartSpecificPosDocking[i + 4] := GVL_CartControlParameters.g_surgicalOrientPos[i_UIData.m_surgicalSite, i_UIData.m_surgicalLocation,i];
	END_IF
END_FOR

m_surgicalStatusF(CLK:= GVL_interactUI.g_surgicalStatus , Q=> );
IF m_surgicalStatusF.Q THEN
	cartDrapingState := 0;
END_IF

IF NOT (m_cartDataFromUI.m_surgicalSite = i_UIData.m_surgicalSite) OR NOT (m_cartDataFromUI.m_surgicalLocation = i_UIData.m_surgicalLocation) THEN
	cartDockingState := 0;
END_IF

m_cartDataFromUI.m_surgicalSite := i_UIData.m_surgicalSite;
m_cartDataFromUI.m_surgicalLocation := i_UIData.m_surgicalLocation;
END_METHOD

PROPERTY status : ST_CartStatus
GET
status := m_cartStatus;
END_GET
END_PROPERTY

METHOD PUBLIC updateCmds : BOOL
VAR_IN_OUT CONSTANT
	i_cartCtrlCmd : ST_SlaveArmCtrlCmds;
END_VAR
VAR
	i:INT;
END_VAR
m_cmdJntTrq:=i_cartCtrlCmd.m_cmdJntTrq;
m_cmdJntPos :=i_cartCtrlCmd.m_cmdJntPos;
m_cmdJntVel :=i_cartCtrlCmd.m_cmdJntVel;


// enable/disable joints
enable(i_cartCtrlCmd.m_jntEnableFlag);

// position/Velocity control
FOR i:=1 TO g_sJntNum DO 
	IF i_cartCtrlCmd.m_jntOPMode[i]=DriverOPMode_Pos THEN
		m_cmdJntTrq[i]:=0;
		m_cmdJntVel[i]:=0;
		m_cartJoints[i].updateCmd(DriverOPMode_Pos,m_cmdJntPos[i],m_cmdJntTrq[i],m_cmdJntVel[i]);
	ELSIF i_cartCtrlCmd.m_jntOPMode[i]=DriverOPMode_Vel THEN
		m_cmdJntTrq[i]:=0;
		m_cmdJntPos[i]:=0;
		m_cartJoints[i].updateCmd(DriverOPMode_Pos,m_cmdJntPos[i],m_cmdJntTrq[i],m_cmdJntVel[i]);
	ELSIF i_cartCtrlCmd.m_jntOPMode[i]=DriverOPMode_MZPos  THEN
		m_cmdJntTrq[i]:=0;
		m_cmdJntVel[i]:=0;
		//Input torque mode because the operating mode word for the contour position mode of the MingZhi driver is 1
		m_cartJoints[i].updateCmd(DriverOPMode_Trq,m_cmdJntPos[i],m_cmdJntTrq[i],m_cmdJntVel[i]);
	ELSIF i_cartCtrlCmd.m_jntOPMode[i]=DriverOPMode_cspMZ  THEN
		 m_cartJoints[i].updateCmd(DriverOPMode_cspMZ,m_cmdJntPos[i],m_cmdJntTrq[i],m_cmdJntVel[i]);
	ELSIF DriverOPMode_csvMZ = i_cartCtrlCmd.m_jntOPMode[i] THEN
		m_cartJoints[i].updateCmd(DriverOPMode_csvMZ,m_cmdJntPos[i],m_cmdJntTrq[i],m_cmdJntVel[i]);
	END_IF
END_FOR

// collision check
m_collisionFlag := m_collisionDetection.run(m_rawJntCurrent, m_cmdJntPos, m_curJntVel);
END_METHOD

METHOD PUBLIC updateStatus : BOOL
VAR_INPUT
END_VAR
VAR
	i:INT;
END_VAR
// update joint data
FOR i:=1 TO g_sJntNum DO
	m_cartJoints[i].updateStatus();
END_FOR

//IO output   Horizontal laser IO output   Cross laser IO output
checkIO();


// get joint data
FOR i:=1 TO g_cartJntNum DO
	m_curMotorPos[i]:=m_cartJoints[i].motorPos;
	m_curLinkPos[i]:=m_cartJoints[i].linkPos;
	m_curLinkSingle[i]:=m_cartJoints[i].linkSingle;
	m_curJntPos[i]:=m_cartJoints[i].jntPos;
	m_curJntVel[i]:=m_cartJoints[i].jntVel;
	m_curJntTrq[i]:=m_cartJoints[i].jntTrq;
	m_rawJntCurrent[i]:=m_cartJoints[i].rawCurrent;
	m_filtJntCurrent[i]:=m_cartJoints[i].filtCurrent;
	m_cmdJntCurrent[i]:=m_cartJoints[i].cmdCurrent;
END_FOR
END_METHOD

END_FUNCTION_BLOCK

// ---- FBs_Auxiliary/FB_trocarDetect.TcPOU
FUNCTION_BLOCK FB_trocarDetect
VAR_INPUT
END_VAR
VAR_OUTPUT
END_VAR
VAR
	m_trocarOnCounts :INT :=0;
	m_trocarOnCountThres :INT :=50;
END_VAR

// check if instrument is on
METHOD run : BOOL
VAR_INPUT
	IOValue :UDINT;
END_VAR
// trocar io is 5th bit 
IF 32=(IOValue AND 10#32) THEN
	m_trocarOnCounts :=MIN(m_trocarOnCounts +1,m_trocarOnCountThres);
ELSE
	m_trocarOnCounts :=0;
END_IF

run := m_trocarOnCounts >= m_trocarOnCountThres;
END_METHOD

END_FUNCTION_BLOCK

// ---- FBs_Auxiliary/FB_rotaButtonDetect.TcPOU
FUNCTION_BLOCK FB_rotaButtonDetect
VAR_INPUT
END_VAR
VAR_OUTPUT
END_VAR
VAR
	m_rotaButtonUpOnCounts :INT :=0;
	m_rotaButtonUpOnCountThres :INT :=50;
	m_rotaButtonDownOnCounts :INT :=0;
	m_rotaButtonDownOnCountThres :INT :=-50;
END_VAR

// check if instrument is on
METHOD run : UDINT
VAR_INPUT
	IOValue :UDINT;
END_VAR
// 
IF 1=(IOValue AND 16#01) OR 2=(IOValue AND 16#02) THEN
	m_rotaButtonUpOnCounts :=MIN(m_rotaButtonUpOnCounts +1,m_rotaButtonUpOnCountThres);
ELSE
	m_rotaButtonUpOnCounts :=0;
END_IF

IF m_rotaButtonUpOnCounts >= m_rotaButtonUpOnCountThres THEN
	run := IOValue;
ELSE
	run := 0;
END_IF
END_METHOD

END_FUNCTION_BLOCK

// ---- FBs_Robots/FB_CartJoint.TcPOU
FUNCTION_BLOCK FB_CartJoint EXTENDS FB_JointBase
VAR_INPUT
END_VAR
VAR_OUTPUT
END_VAR
VAR
	//Cart motor output IO
	m_cartMotorOutput AT %Q*	:ST_CartMotorOutput;
	
	m_cmdAcc:LREAL;
	
END_VAR

METHOD cmd2motorMZ : DINT
VAR_INPUT
	i_cmd:LREAL;
	i_controlCycleTime :LREAL;
END_VAR
cmd2motorMZ:=LREAL_TO_DINT(((4*m_motorEncoderRes*m_motorReduction*i_controlCycleTime)/(2*pi))*i_cmd*65536);
END_METHOD

METHOD PUBLIC enableMZ : BOOL
VAR_INPUT
END_VAR
IF (MZDriverStatusWord_SwitchOnDisable AND m_motorInputs.m_statusWord) = MZDriverStatusWord_SwitchOnDisable    THEN
	m_motorOutputs.m_controlWord:=DriverCtrlWord_INIT;
	enableMZ := FALSE;
ELSIF (MZDriverStatusWord_OperationEnbale AND m_motorInputs.m_statusWord) = MZDriverStatusWord_OperationEnbale THEN
	enableMZ :=  TRUE;
ELSIF (MZDriverStatusWord_SwitchOn AND m_motorInputs.m_statusWord) =  MZDriverStatusWord_SwitchOn THEN
	m_motorOutputs.m_controlWord:=DriverCtrlWord_OP;
	enableMZ :=  FALSE;
ELSIF (MZDriverStatusWord_ReadyToSwitchOn AND m_motorInputs.m_statusWord) = MZDriverStatusWord_ReadyToSwitchOn THEN
	m_motorOutputs.m_controlWord:=DriverCtrlWord_PREOP;
	enableMZ :=  FALSE;
ELSIF (MZDriverStatusWord_Fault AND m_motorInputs.m_statusWord) = MZDriverStatusWord_Fault THEN
	m_motorOutputs.m_controlWord:=DriverCtrlWord_FaultReset;
//ELSE
//	m_motorOutputs.m_controlWord:=DriverCtrlWord_INIT;
//	enable :=  FALSE;
END_IF
END_METHOD

METHOD PUBLIC init : BOOL
VAR_INPUT
	i_jntIdx :INT;
	i_controlCycleTime :LREAL;
END_VAR
m_jntIdx:=i_jntIdx;
m_cycleTime := i_controlCycleTime;

// hardware parameters
m_motorEncoderRes :=GVL_CartMotorParameters.g_incEncoderRes[i_jntIdx];
m_linkEncoderRes :=GVL_CartMotorParameters.g_absEncoderRes[i_jntIdx];
m_motorReduction :=GVL_CartMotorParameters.g_motorReduction[i_jntIdx];
m_linkEncoderReduction :=GVL_CartMotorParameters.g_absEncoderReduction[i_jntIdx];
m_trqConst :=GVL_CartMotorParameters.g_motorTrqConst[i_jntIdx];
m_maxCurrent :=GVL_CartMotorParameters.g_motorMaxCurrent[i_jntIdx];
m_motorDir :=GVL_CartMotorParameters.g_motorDir[i_jntIdx];								
m_minJntPos	:=GVL_CartMotorParameters.g_minJntPos[i_jntIdx];
m_maxJntPos	:=GVL_CartMotorParameters.g_maxJntPos[i_jntIdx];

//link encoder calibartion data
m_linkEncoderDir :=GVL_CartJointEncoderCaliData.g_asbEncoderDir[i_jntIdx];
m_minLinkEncoder :=GVL_CartJointEncoderCaliData.g_minLinkEncoder[ i_jntIdx] - m_linkEncoderDir*GVL_SetupJointEncoderCaliData.g_linkEncLimitBuffer; // expand limit
m_maxLinkEncoder :=GVL_CartJointEncoderCaliData.g_maxLinkEncoder[ i_jntIdx] + m_linkEncoderDir*GVL_SetupJointEncoderCaliData.g_linkEncLimitBuffer; // expand limit
m_caliLinkEncoder :=GVL_CartJointEncoderCaliData.g_caliLinkEncoder[ i_jntIdx];
m_linkEncCaliJntPos :=GVL_CartJointEncoderCaliData.g_linkEncCaliJntPos[i_jntIdx];
m_linkEncZeroCross :=GVL_CartJointEncoderCaliData.g_linkEncZeroCross[ i_jntIdx];
m_multiCycles :=GVL_CartJointEncoderCaliData.g_multipleCyclesJoint[i_jntIdx];

// convert cali link encoder if joint cross zero
IF 1=m_linkEncZeroCross THEN
	IF 1=m_linkEncoderDir AND m_caliLinkEncoder < m_minLinkEncoder THEN
		m_caliLinkEncoder := GVL_CartJointEncoderCaliData.g_caliLinkEncoder[ i_jntIdx] + m_linkEncoderRes;
	ELSIF -1=m_linkEncoderDir AND m_caliLinkEncoder < m_maxLinkEncoder THEN
		m_caliLinkEncoder := GVL_CartJointEncoderCaliData.g_caliLinkEncoder[ i_jntIdx] + m_linkEncoderRes;
	END_IF
END_IF

// macro data
m_trq2CurrentRatio:=m_motorDir * 1000.0/(m_trqConst*m_motorReduction);
m_current2TrqRatio:=m_motorDir * (m_trqConst*m_motorReduction)/1000.0;
m_linkEnc2PosRatio := 2*PI*m_linkEncoderDir/(m_linkEncoderReduction*m_linkEncoderRes);
m_motorEnc2PosRatio := 2*PI * m_motorDir/(m_motorReduction * m_motorEncoderRes);


// motor data init
m_rawJntVel :=0;
m_curJntVel:=0;
m_curJntTrq :=0;
m_rawCurrent :=0;
m_filtCurrent :=0;
m_cmdJntVel :=0.0;
m_cmdJntTrq :=0.0;
m_cmdCurrent := 0.0;

// filter init
m_jntVelLpf.init(1, GVL_CartControlParameters.g_curJntVelLpfCutoffFreq, g_cartCtrlFreq);
m_cmdTrqLpf.init(1, GVL_CartControlParameters.g_cmdJntTrqLpfCutoffFreq, g_cartCtrlFreq);
m_curTrqLpf.init(1, GVL_CartControlParameters.g_curJntTrqLpfCutoffFreq, g_cartCtrlFreq);

// driver init value
m_motorOutputs.m_controlWord:=DriverCtrlWord_INIT;
m_motorOutputs.m_opMode:=INT_TO_SINT(DriverOPMode_Pos);
m_motorOutputs.m_cmdCurrent:=0;
m_motorOutputs.m_cmdMotorEncoder:=m_motorInputs.m_motorEncoder;
END_METHOD

METHOD PUBLIC updateCmd : BOOL
VAR_INPUT
	i_opMode : E_DriverOPMode;
	i_cmdPos :LREAL;
	i_cmdTrq :LREAL;
	i_cmdVel :LREAL;
END_VAR
VAR
	i:INT;
END_VAR
m_motorOutputs.m_opMode:=INT_TO_SINT( i_opMode);

// pos mode
IF i_opMode = DriverOPMode_Pos OR i_opMode = DriverOPMode_cspMZ  THEN
	m_motorOutputs.m_cmdCurrent:=0;
	m_cmdJntPos :=i_cmdPos;
	m_motorOutputs.m_cmdMotorEncoder :=motorPos2Enc(m_cmdJntPos);
ELSIF i_opMode = DriverOPMode_Vel THEN
	m_cmdJntVel := i_cmdVel;
	m_cartMotorOutput.m_cmdVelMzVelMode := cmd2motorMZ(m_cmdJntVel, g_cartCtrlCycleTime);
ELSIF i_opMode = DriverOPMode_Trq THEN   //Here the torque mode is equal to the contour position mode of the MingZhi driver
	m_cmdJntVel := i_cmdVel;
	m_cmdAcc:=i_cmdVel*2;
	m_cmdJntPos:=i_cmdPos;
	m_cartMotorOutput.m_cmdAccMz :=cmd2motorMZ(m_cmdAcc, g_cartCtrlCycleTime);
	m_cartMotorOutput.m_cmdVelMz := cmd2motorMZ(m_cmdJntVel, g_cartCtrlCycleTime);
	m_motorOutputs.m_cmdMotorEncoder := motorPos2Enc(m_cmdJntVel);
ELSIF i_opMode = DriverOPMode_csvMZ THEN
	m_cmdJntVel := i_cmdVel;
	m_cartMotorOutput.m_cmdVelMzVelMode := cmd2motorMZ(m_cmdJntVel, g_cartCtrlCycleTime);
END_IF
END_METHOD

METHOD PUBLIC updateStatus : BOOL
VAR_INPUT
END_VAR
// compute joint position
m_curLinkPos:= linkEnc2Pos();
m_curMotorPos:=motorEnc2Pos();
m_curLinkSingle := m_curLinkPos - 2*PI* m_linkEncCycles;

// Cart joint1-4 have no link enconder, use motor position
IF m_jntIdx <= 4 THEN
	m_curJntPos := m_curMotorPos;
ELSE
	m_curJntPos := m_curLinkPos;
END_IF

// compute joint velocity
m_curVelCalCycles := m_curVelCalCycles+1;
IF m_curVelCalCycles > m_velCalcCycles THEN
	m_rawJntVel:= (m_curJntPos-m_lastJntPos)/(m_cycleTime*m_velCalcCycles);
	m_curJntVel := m_jntVelLpf.run(m_rawJntVel);
	m_lastJntPos :=m_curJntPos;	
	m_curVelCalCycles:=1;
END_IF


// current and torque
m_rawCurrent := m_motorInputs.m_current;
m_filtCurrent := m_curTrqLpf.run(m_rawCurrent);
m_curJntTrq := m_filtCurrent * m_current2TrqRatio;
END_METHOD

END_FUNCTION_BLOCK

// ---- FBs_Robots/FB_JointBase.TcPOU
FUNCTION_BLOCK FB_JointBase
VAR_INPUT
END_VAR
VAR_OUTPUT
END_VAR
VAR
	// arm and joint index
	m_armIdx :INT;
	m_jntIdx :INT;
	
	// motor IO
	m_motorInputs AT%I*	:ST_MotorInputs;
	m_motorOutputs AT%Q* :ST_MotorOutputs;
	
	// cycle time
	m_cycleTime :LREAL;
	
	// calibrated link encoder data
	m_minLinkEncoder :DINT;
	m_maxLinkEncoder :DINT;
	m_caliLinkEncoder :DINT;
	m_linkEncCaliJntPos :LREAL;
	m_linkEncZeroCross :INT;
	m_initMotorEnc : DINT;
	m_multiCycles :INT;
	
	// joint position from link encoder after power on
	m_initLinkPos :LREAL;
	
	// data for link encoder multiple cycles
	m_lastLinkEncoder :DINT;
	m_linkEncCycles:INT;
	
	// device paramters
	m_motorEncoderRes :DINT;
	m_linkEncoderRes :DINT;
	m_motorReduction :LREAL;
	m_linkEncoderReduction :LREAL;
	m_trqConst :LREAL;
	m_maxCurrent :LREAL;
	m_motorDir :INT;								
	m_linkEncoderDir :INT;
	m_minJntPos: LREAL;
	m_maxJntPos: LREAL;
	
	// macro defined data for quick calculation
	m_trq2CurrentRatio:LREAL;
	m_current2TrqRatio:LREAL;
	m_linkEnc2PosRatio :LREAL;
	m_motorEnc2PosRatio :LREAL;
	
	// joint data
	m_curMotorPos :LREAL;
	m_curLinkPos :LREAL;
	m_curLinkSingle :LREAL;//[0-360]
	m_curJntPos	:LREAL;
	m_curJntVel :LREAL;
	m_rawJntVel :LREAL;
	m_curJntTrq :	LREAL;
	m_rawCurrent : LREAL;
	m_filtCurrent : LREAL;
	m_cmdJntPos :LREAL;
	m_cmdJntVel :LREAL;
	m_cmdJntTrq :LREAL;
	m_cmdCurrent : LREAL;
	m_lastJntPos :LREAL;
	
	// velocity filter
	m_jntVelLpf :FB_LowPassFilter;
	
	// command torque filter
	m_curTrqLpf : FB_LowPassFilter;
	m_cmdTrqLpf :FB_LowPassFilter;
	
	// velocity is calculated every (m_velCalcCycles) control cycles
	// TODO: insturment joint motor can not reach 4k now, so calculate their velocity with 1k frequency, need to remove later
	m_velCalcCycles :INT :=1;
	m_curVelCalCycles :INT :=1;
	
	// SDO writer
	m_opModeSDOWrite:FB_EcCoESdoWrite;
	m_MotorCurrentSDOWrite:FB_EcCoESdoWrite;
	
END_VAR

PROPERTY cmdCurrent : LREAL
GET
cmdCurrent:=m_cmdCurrent;
END_GET
END_PROPERTY

METHOD PUBLIC disable : BOOL
VAR_INPUT
END_VAR
m_motorOutputs.m_controlWord:=DriverCtrlWord_INIT;
disable:=true;
END_METHOD

PROPERTY driveInput : ST_MotorInputs
GET
driveInput := m_motorInputs;
END_GET
END_PROPERTY

PROPERTY driveOutput : ST_MotorOutputs
GET
driveOutput := m_motorOutputs;
END_GET
END_PROPERTY

METHOD PUBLIC enable : BOOL
VAR_INPUT
END_VAR
IF DriverStatusWord_INIT = m_motorInputs.m_statusWord THEN
	m_motorOutputs.m_controlWord:=DriverCtrlWord_PREOP;
	enable := FALSE;
ELSIF DriverStatusWord_PREOP = m_motorInputs.m_statusWord THEN
	m_motorOutputs.m_controlWord:=DriverCtrlWord_OP;
	enable :=  FALSE;
ELSIF DriverStatusWord_OP = m_motorInputs.m_statusWord THEN
	enable :=  TRUE;
//ELSE
//	m_motorOutputs.m_controlWord:=DriverCtrlWord_INIT;
//	enable :=  FALSE;
END_IF
END_METHOD

PROPERTY filtCurrent : LREAL
GET
filtCurrent:=m_filtCurrent;
END_GET
END_PROPERTY

METHOD PUBLIC initJntPos : BOOL
VAR_INPUT
END_VAR
m_lastLinkEncoder :=m_motorInputs.m_linkEncoder;
m_linkEncCycles:=0;
m_curLinkPos :=linkEnc2Pos();
m_initLinkPos:=m_curLinkPos;
m_initMotorEnc :=m_motorInputs.m_motorEncoder;
m_curMotorPos:=motorEnc2Pos();
m_curJntPos := m_curMotorPos;
m_cmdJntPos :=m_curJntPos;	
m_lastJntPos :=m_curJntPos;
END_METHOD

PROPERTY initLinkPos : lreal
GET
initLinkPos:=m_initLinkPos;
END_GET
SET
m_initLinkPos:=initLinkPos;
END_SET
END_PROPERTY

METHOD PUBLIC isEnabled : BOOL
VAR_INPUT
END_VAR
isEnabled :=(DriverStatusWord_OP = m_motorInputs.m_statusWord);
END_METHOD

PROPERTY jntPos : LREAL
GET
jntPos := m_curJntPos;
END_GET
END_PROPERTY

PROPERTY jntTrq : LREAL
GET
jntTrq:=m_curJntTrq;
END_GET
END_PROPERTY

PROPERTY jntVel : LREAL
GET
jntVel := m_curJntVel;
END_GET
END_PROPERTY

METHOD PROTECTED linkEnc2Pos : LREAL
VAR_INPUT
END_VAR
VAR
	incLinkPos :LREAL;
	newLinkEnc :DINT;
END_VAR
// cycle check
IF 1=m_multiCycles THEN
	IF (m_motorInputs.m_linkEncoder - m_lastLinkEncoder)*m_linkEncoderDir < -m_linkEncoderRes/2 THEN
		m_linkEncCycles :=m_linkEncCycles+1;
	ELSIF (m_motorInputs.m_linkEncoder - m_lastLinkEncoder)*m_linkEncoderDir > m_linkEncoderRes/2 THEN
		m_linkEncCycles :=m_linkEncCycles-1;
	END_IF
END_IF
m_lastLinkEncoder:=m_motorInputs.m_linkEncoder;

// convert link encoder if joint cross zero
newLinkEnc := m_motorInputs.m_linkEncoder;
IF 1=m_linkEncZeroCross AND 0 = m_multiCycles THEN
	IF 1=m_linkEncoderDir AND m_motorInputs.m_linkEncoder < m_minLinkEncoder THEN
		newLinkEnc := m_motorInputs.m_linkEncoder + m_linkEncoderRes;
	ELSIF -1=m_linkEncoderDir AND m_motorInputs.m_linkEncoder < m_maxLinkEncoder THEN
		newLinkEnc := m_motorInputs.m_linkEncoder + m_linkEncoderRes;
	END_IF
END_IF

// motion from calibrated points
incLinkPos := (newLinkEnc-m_caliLinkEncoder)*m_linkEnc2PosRatio;

// absolute joint position
linkEnc2Pos := incLinkPos + m_linkEncCaliJntPos + 2*PI* m_linkEncCycles;
END_METHOD

PROPERTY PUBLIC linkPos : LREAL
GET
linkPos:=m_curLinkPos;
END_GET
END_PROPERTY

PROPERTY linkSingle : LREAL
GET
linkSingle :=m_curLinkSingle;
END_GET
END_PROPERTY

METHOD PROTECTED motorEnc2Pos : LREAL
VAR_INPUT
END_VAR
motorEnc2Pos:= (m_motorInputs.m_motorEncoder-m_initMotorEnc)* m_motorEnc2PosRatio +m_initLinkPos;
END_METHOD

PROPERTY PUBLIC motorPos : LREAL
GET
motorPos := m_curMotorPos;
END_GET
END_PROPERTY

METHOD PROTECTED motorPos2Enc : DINT
VAR_INPUT
	i_jntPos :LREAL;
END_VAR

VAR
END_VAR
motorPos2Enc := LREAL_TO_DINT((i_jntPos-m_initLinkPos)/m_motorEnc2PosRatio + m_initMotorEnc);
END_METHOD

PROPERTY rawCurrent : LREAL
GET
rawCurrent := m_rawCurrent;
END_GET
END_PROPERTY

METHOD PROTECTED singleCyclePos : LREal
VAR_INPUT
END_VAR
VAR
	cycles :lreal;
END_VAR
cycles := ABS(FLOOR( m_curJntPos/g_2pi));
IF m_curJntPos<0 THEN
	singleCyclePos := m_curJntPos+cycles*g_2pi;
ELSE
	singleCyclePos := m_curJntPos-cycles*g_2pi;
END_IF
END_METHOD

METHOD PUBLIC updateCmds : BOOL
VAR_INPUT
	i_opMode : E_DriverOPMode;
	i_cmdPos :LREAL;
	i_cmdTrq :LREAL;
END_VAR
VAR
	filtCmdTrq :LREAL;
END_VAR
m_motorOutputs.m_opMode:=INT_TO_SINT( i_opMode);
// pos mode
IF i_opMode = DriverOPMode_Pos THEN
	m_motorOutputs.m_cmdCurrent:=0;
	m_cmdTrqLpf.reset();	
//	i_cmdPos:=LIMIT(m_minJntPos, i_cmdPos, m_maxJntPos); // May cause position jump, Do this in safety check. 
	m_cmdJntPos :=i_cmdPos;
	m_motorOutputs.m_cmdMotorEncoder :=motorPos2Enc(m_cmdJntPos);
ELSIF i_opMode = DriverOPMode_Trq THEN
	filtCmdTrq:=m_cmdTrqLpf.run(i_cmdTrq);
	m_motorOutputs.m_cmdCurrent:=LREAL_TO_DINT(LIMIT(-m_maxCurrent, filtCmdTrq*m_trq2CurrentRatio,m_maxCurrent));
	m_motorOutputs.m_cmdMotorEncoder :=m_motorInputs.m_motorEncoder; 
END_IF
m_cmdCurrent:=m_motorOutputs.m_cmdCurrent;
END_METHOD

METHOD PUBLIC updateStatus : BOOL
VAR_INPUT
END_VAR
// compute joint position
m_curLinkPos:= linkEnc2Pos();
m_curMotorPos:=motorEnc2Pos();
m_curJntPos := m_curMotorPos;
m_curLinkSingle := singleCyclePos();

// compute joint velocity
m_curVelCalCycles := m_curVelCalCycles+1;
IF m_curVelCalCycles > m_velCalcCycles THEN
	m_rawJntVel:= (m_curJntPos-m_lastJntPos)/(m_cycleTime*m_velCalcCycles);
	m_curJntVel := m_jntVelLpf.run(m_rawJntVel);
	m_lastJntPos :=m_curJntPos;	
	m_curVelCalCycles:=1;
END_IF


// current and torque
m_rawCurrent := m_motorInputs.m_current;
m_filtCurrent := m_curTrqLpf.run(m_rawCurrent);
m_curJntTrq := m_filtCurrent * m_current2TrqRatio;
END_METHOD

END_FUNCTION_BLOCK

// ---- FBs_Auxiliary/FB_cartJntEnableDetect.TcPOU
FUNCTION_BLOCK FB_cartJntEnableDetect
VAR_INPUT
END_VAR
VAR_OUTPUT
END_VAR
VAR
	m_jntEnableCounts :INT :=0;
	m_jntEnableCountThres :INT :=100;
END_VAR

// check if instrument is on
METHOD run : BOOL
VAR_INPUT
	IOValue :BOOL;
END_VAR
// trocar io is 5th bit 
IF TRUE=IOValue THEN
	m_jntEnableCounts :=MIN(m_jntEnableCounts +1,m_jntEnableCountThres);
ELSE
	m_jntEnableCounts :=0;
END_IF

run := m_jntEnableCounts >= m_jntEnableCountThres;
END_METHOD

END_FUNCTION_BLOCK

// ---- FBs_Auxiliary/FB_cartJntDisenableDetect.TcPOU
FUNCTION_BLOCK FB_cartJntDisenableDetect
VAR_INPUT
END_VAR
VAR_OUTPUT
END_VAR
VAR
	m_jntEnableCounts :INT :=0;
	m_jntEnableCountThres :INT :=100;
END_VAR

// check if instrument is on
METHOD run : BOOL
VAR_INPUT
	IOValue :BOOL;
END_VAR
// trocar io is 5th bit 
IF TRUE=IOValue THEN
	m_jntEnableCounts :=MIN(m_jntEnableCounts +1,m_jntEnableCountThres);
ELSE
	m_jntEnableCounts :=0;
END_IF

run := m_jntEnableCounts >= m_jntEnableCountThres;
END_METHOD

END_FUNCTION_BLOCK

// ---- Mains/SafetyCheck.TcPOU
PROGRAM SafetyCheck
VAR
	// slave robot information, including arm status and cartesian data
	m_slaveStatus AT %I* :ST_slaveStatus;
	
	// slave robot joint data
	m_slaveJointData AT %I* :ST_slaveJointData;
	
	// setup robot information
	m_setupStatus AT %I* :ST_SetupStatus;
	
	// setup robot joint data
	m_setupJointsData AT %I* :ST_SetupJointData;
	
	// master robot data, input from master controller box
	m_masterRobotData AT %I* : MSCommu_MasterStatus;
	
	// error check result
	m_safetyCheckData AT %Q* :ST_SafetyData;
	
	// Output cart status
	m_cartStatus AT%I* : ST_CartStatus;
	
	// cart joint data
	m_cartJointsData AT %I* :ST_CartJointData;
	
	//emergency stop and stop botton
	m_stopButton AT %I*: BOOL;
	m_emergencyStopButton AT %I*: BOOL;
	
	//warning tone
	m_warningTone AT %Q*:ARRAY [1..4] OF BOOL;
	
	m_initFlag:bool;
	
	m_SafetyCheck : Fb_SafetyCheck;
	m_checkVariable : ARRAY[1..g_maxNum] OF checkInputVariable;
	m_EtherCATCheck :ARRAY [1..g_maxNum,1..g_maxArmJoint] OF Fb_EtherCATCheck;
	m_errCode :ARRAY [1..3] OF UDINT;
	i , j: INT;
	
	//error robot data record
	m_dataRecord : Fb_dataRecord;
	
	// original position of remote center point when fisrt enter hold state
	m_dsrRcpPos :ARRAY[1..g_sArmNum] OF Vec3d;
	m_rcpPosErrCounts :ARRAY[1..g_sArmNum] OF INT := [4(0)];
	m_rcpPosErr :ARRAY[1..g_sArmNum] OF Vec3d;		// rcp position error
	m_curJntPosLast : ARRAY [1..g_maxArmNum] OF vec13di;  
	m_armErrCodeRefreshLast : ARRAY [1..4] OF UINT;
	
	m_armsRS:ARRAY [1..g_maxArmNum,1..30] OF RS;//复位优先双稳态器
	m_cartRS:ARRAY [1..30] OF RS;//复位优先双稳态器
	m_scopeArmNoReady : BOOL;
	m_joysticksTrigger : BOOL;
	// wait time before robot init  for ethercat to be statble 
	m_safetyCheckInitWaitTime : LREAL:=0;
END_VAR

// reset data
IF FALSE = m_initFlag  THEN
	FOR i:=1  TO g_sArmNum DO 
		m_safetyCheckData.m_slaveErrFlag[i]:=FALSE;
		m_safetyCheckData.m_setupErrFlag[i]:=FALSE;
		m_safetyCheckData.m_cartErrFlag:=FALSE;
	END_FOR
	m_initFlag:=TRUE;
END_IF

armSafetyCheckInputCast();

armSafetyCheckAllowed();

robotPromptMassageCast();

// wait communication to be stable
IF(m_safetyCheckInitWaitTime<g_robotSafetyCheckWaitTime) THEN
	m_safetyCheckInitWaitTime := m_safetyCheckInitWaitTime+g_setupArmCtrlCycleTime;
	RETURN;
END_IF


FOR i:=1  TO g_maxNum DO
	m_SafetyCheck.systemSafetyCheck(i,m_checkVariable,m_cartJointsData,m_setupJointsData,m_slaveJointData);
END_FOR


//error flag to control
readErrFlag();

//Fault code for UI
m_SafetyCheck.errCodeUpdating();

//The fault code is sent to the UI
GVL_interactUI.g_errIdType3:=m_SafetyCheck.o_ErrCode[3];
GVL_interactUI.g_errIdType2:=m_SafetyCheck.o_ErrCode[2];
GVL_interactUI.g_errIdType1:=m_SafetyCheck.o_ErrCode[1];
GVL_interactUI.g_popupErrorArm1 := m_SafetyCheck.m_armErrCodePopup[1];
GVL_interactUI.g_popupErrorArm2 := m_SafetyCheck.m_armErrCodePopup[2];
GVL_interactUI.g_popupErrorArm3 := m_SafetyCheck.m_armErrCodePopup[3];
GVL_interactUI.g_popupErrorArm4 := m_SafetyCheck.m_armErrCodePopup[4];
FOR i:=1  TO g_sArmNum DO
	IF m_SafetyCheck.m_armErrCodeRefresh[i] <> m_armErrCodeRefreshLast[i] THEN
		GVL_interactUI.g_popupRefresh[i] := 1;
	END_IF
	m_armErrCodeRefreshLast[i] := m_SafetyCheck.m_armErrCodeRefresh[i];
END_FOR

//clear fault
IF GVL_interactUI.g_uiFaultReset=1 OR m_masterRobotData.m_uiResetFault = 1 THEN
	m_SafetyCheck.errFlagReset();
	GVL_interactUI.g_uiFaultReset := 0;
END_IF

//robot record information
m_dataRecord.run(m_checkVariable , m_cartStatus , m_cartJointsData , m_setupStatus , m_slaveStatus , m_setupJointsData , m_slaveJointData );

m_warningTone := warningTone();

METHOD armSafetyCheckAllowed : BOOL
VAR_INPUT
END_VAR
VAR
	i , j : INT; 
END_VAR
FOR i := 1 TO g_maxArmNum DO
	FOR j := 1 TO g_maxArmJoint DO
		IF j > 5 THEN
			//fault code 16#3003 
			m_SafetyCheck.checkPermit[i].m_linkEncErr[j] := m_checkVariable[i].m_slaveDriverInput[j-g_setupJntNum].m_statusWord<>0;
			//fault code 16#3002 
			m_SafetyCheck.checkPermit[i].m_currentIsNotUpdate[j] :=m_checkVariable[i].m_slaveDriverInput[j-g_setupJntNum].m_statusWord<>0 ;
			//fault code 16#2002
			m_SafetyCheck.checkPermit[i].m_armJntFollowErr[j] := m_checkVariable[i].m_slaveDriverInput[j-g_setupJntNum].m_statusWord = DriverStatusWord_OP ;
			//fault code 16#200B
			m_SafetyCheck.checkPermit[i].m_jntCurrentCtrlErr[j] := m_checkVariable[i].m_slaveDriverOutput[j-g_setupJntNum].m_opMode = DriverOPMode_Trq;
		ELSE
			//fault code 16#3003 
			m_SafetyCheck.checkPermit[i].m_linkEncErr[j] := m_checkVariable[i].m_setupDriverInput[j].m_statusWord<>0;
			//fault code 16#3002
			m_SafetyCheck.checkPermit[i].m_currentIsNotUpdate[j] := m_checkVariable[i].m_setupDriverInput[j].m_statusWord<>0 AND j > 2;
			//fault code 16#2002
			m_SafetyCheck.checkPermit[i].m_armJntFollowErr[j] := m_checkVariable[i].m_setupDriverInput[j].m_statusWord = DriverStatusWord_OP AND j > 2;
			//fault code 16#200B
			m_SafetyCheck.checkPermit[i].m_jntCurrentCtrlErr[j] := m_checkVariable[i].m_setupDriverOutput[j].m_opMode = DriverOPMode_Trq AND j > 2;
			
		END_IF
		//fault code 16#3002
		m_SafetyCheck.checkPermit[i].m_jntStatusErr[j] := TRUE;
		//fault code 16#3004
		m_SafetyCheck.checkPermit[i].m_driveErr[j] := TRUE;
		//fault code 16#3005
		m_SafetyCheck.checkPermit[i].m_armJntEncErr[j] := TRUE;
		//fault code 16#3006
		m_SafetyCheck.checkPermit[i].m_outOfLimit[j] := TRUE;
		//fault code 16#3008
		m_SafetyCheck.checkPermit[i].m_motPhieErr[j] := TRUE;
		//fault code 16#2003
		m_SafetyCheck.checkPermit[i].m_jntVelErr[j] := TRUE;
		//fault code 16#2004
		m_SafetyCheck.checkPermit[i].m_spacePoseErr[j] := m_slaveStatus.m_armState[i] = SlaveArmState_MasterSlave AND  norm(m_slaveStatus.m_masterSlavePoseError[i])<g_smallNum;
		//fault code 16#2005
		m_SafetyCheck.checkPermit[i].m_jntCurrentErr[j] := TRUE;
		//fault code 16#2007
		m_SafetyCheck.checkPermit[i].m_fixedPointErr := m_slaveStatus.m_armState[i] = SlaveArmState_MasterSlave;
		//fault code 16#2008
		m_SafetyCheck.checkPermit[i].m_cmdJntSaltation[j] := m_slaveStatus.m_armState[i] = SlaveArmState_MasterSlave;
		//fault code 16#200F
		m_SafetyCheck.checkPermit[i].m_instruOpenAngle := FALSE;
	END_FOR
END_FOR
END_METHOD

METHOD armSafetyCheckInputCast : BOOL
VAR_INPUT
END_VAR

VAR
	i , j: INT; 
END_VAR
FOR i := 1 TO g_maxArmNum DO
	//emergency stop 、stop button and ui stop 
	m_checkVariable[i].EmergencyStop := m_emergencyStopButton;
	m_checkVariable[i].PCStopButton := GVL_interactUI.g_stopButtonFormUI;
	m_checkVariable[i].SlaveStopButton := m_stopButton;
	m_checkVariable[i].MasterStopButton := m_masterRobotData.m_masterStopButton;
	
	IF m_setupStatus.m_armState[i] <> SetupArmState_Hold THEN
		m_dsrRcpPos[i] := m_setupStatus.m_rcPos[i];
	END_IF
	m_checkVariable[i].m_rcpCheck := m_SafetyCheck.rcpErrCheck(m_dsrRcpPos[i],  m_setupStatus.m_rcPos[i], m_rcpPosErrCounts[i] ,m_rcpPosErr[i]);
	m_checkVariable[i].m_spacePoseErr := m_SafetyCheck.poseErrCheck(m_slaveStatus.m_cmdArmPose[i], m_slaveStatus.m_simArmPose[i] );
	
	//slave robot input cast
	FOR j:=1 TO  g_sJntNum DO 		
		m_checkVariable[i].m_slaveDriverInput[j] := SlaveArmControl.m_slaveRobot.m_slaveArms[i].m_joints[j].m_motorInputs;
		//3 joint drive error word at number 6 , move one bit to the right to align with the other joints
		IF j = 3 THEN
			m_checkVariable[i].m_slaveDriverInput[j].m_driverError := SHR(SlaveArmControl.m_slaveRobot.m_slaveArms[i].m_joints[j].m_motorInputs.m_driverError,1);
		END_IF
		m_checkVariable[i].m_slaveDriverOutput[j] := SlaveArmControl.m_slaveRobot.m_slaveArms[i].m_joints[j].m_motorOutputs;
		m_checkVariable[i].m_EtherCATState[j+g_setupJntNum] := m_EtherCATCheck[i,j+g_setupJntNum].EtherCATVerify(GVL_SlaveJointEncoderCaliData.g_slaveArmNetID[i],g_JointNetPort[j+g_setupJntNum]);
		m_checkVariable[i].m_motorEncoderSaltaValue[j+g_setupJntNum] := ABS(m_checkVariable[i].m_slaveDriverInput[j+g_setupJntNum].m_motorEncoder - m_curJntPosLast[i][j+g_setupJntNum]);
		m_curJntPosLast[i][j+g_setupJntNum] := m_checkVariable[i].m_slaveDriverInput[j+g_setupJntNum].m_motorEncoder;
	END_FOR
	
	//setup robot input cast
	FOR j:=1 TO  g_setupJntNum DO 		
		m_checkVariable[i].m_setupDriverInput[j] := SetupArmControl.m_setupRobot.m_setupArms[i].m_joints[j].m_motorInputs;
		m_checkVariable[i].m_setupDriverOutput[j] := SetupArmControl.m_setupRobot.m_setupArms[i].m_joints[j].m_motorOutputs;
		m_checkVariable[i].m_EtherCATState[j] := m_EtherCATCheck[i,j].EtherCATVerify(GVL_SlaveJointEncoderCaliData.g_slaveArmNetID[i],g_JointNetPort[j]);
		m_checkVariable[i].m_motorEncoderSaltaValue[j] := m_checkVariable[i].m_setupDriverInput[j].m_motorEncoder - m_curJntPosLast[i][j];
		m_curJntPosLast[i][j] := m_checkVariable[i].m_setupDriverInput[j].m_motorEncoder;
	END_FOR

END_FOR

//setup robot in-out variable cast
FOR j:=1 TO  g_cartJntNum DO
	m_checkVariable[5].EmergencyStop := m_emergencyStopButton;
	m_checkVariable[5].PCStopButton := GVL_interactUI.g_stopButtonFormUI;
	m_checkVariable[5].SlaveStopButton := m_stopButton;
	m_checkVariable[5].m_cartDriverInput[j] := CartControl.m_cartRobot.m_slaveCart.m_cartJoints[j].m_motorInputs;
	m_checkVariable[5].m_cartDriverOutput[j] := CartControl.m_cartRobot.m_slaveCart.m_cartJoints[j].m_motorOutputs;
	m_checkVariable[5].m_cartEtherCATState[j] := m_EtherCATCheck[5,j].EtherCATVerify(GVL_CartJointEncoderCaliData.g_slaveCartNetID,GVL_CartJointEncoderCaliData.g_slaveCartJointNetPort[j]);
END_FOR
END_METHOD

METHOD joystickAdjust : BOOL
VAR_IN_OUT CONSTANT
	i_joystickValue : vec8d;
END_VAR

VAR
	i : INT;
END_VAR

FOR i := 1 TO 4 DO
	IF 492 > i_joystickValue[i] OR i_joystickValue[i] > 532 THEN
		joystickAdjust := TRUE;
		EXIT;
	END_IF
END_FOR
END_METHOD

METHOD readErrFlag : BOOL
VAR_INPUT
END_VAR
FOR i:=1  TO g_sArmNum DO
	m_safetyCheckData.m_slaveErrFlag[i] := m_SafetyCheck.m_armErrFlag[i,2] OR m_SafetyCheck.m_armErrFlag[i,3];
	m_safetyCheckData.m_setupErrFlag[i] := m_SafetyCheck.m_armErrFlag[i,2] OR m_SafetyCheck.m_armErrFlag[i,3];
END_FOR


GVL_interactUI.g_slaveRecoverErrFlag := BOOL_TO_INT((m_SafetyCheck.m_armErrFlag[1,2] OR m_SafetyCheck.m_armErrFlag[2,2] OR m_SafetyCheck.m_armErrFlag[3,2] OR m_SafetyCheck.m_armErrFlag[4,2]
														OR m_SafetyCheck.m_armErrFlag[g_cartNum,2] OR m_SafetyCheck.m_jntErrFlag[g_cartNum,0,2]) AND GVL_interactUI.g_slaveRunAlone) ;

//cart error flag
m_safetyCheckData.m_cartErrFlag := m_SafetyCheck.m_armErrFlag[g_cartNum,2] OR m_SafetyCheck.m_armErrFlag[g_cartNum,3];
//cart stead foot error flag
m_safetyCheckData.m_cartSteadyFootErr := m_SafetyCheck.m_jntErrFlag[g_cartNum,1,2] OR m_SafetyCheck.m_jntErrFlag[g_cartNum,1,3] 
																	OR m_SafetyCheck.m_jntErrFlag[g_cartNum,2,2] OR m_SafetyCheck.m_jntErrFlag[g_cartNum,2,3] OR m_SafetyCheck.m_jntErrFlag[g_cartNum,0,2];
//cart wheel error flag
m_safetyCheckData.m_cartWheelErr := m_SafetyCheck.m_jntErrFlag[g_cartNum,3,2] OR m_SafetyCheck.m_jntErrFlag[g_cartNum,3,3]
																OR m_SafetyCheck.m_jntErrFlag[g_cartNum,4,2] OR m_SafetyCheck.m_jntErrFlag[g_cartNum,4,3] OR m_SafetyCheck.m_jntErrFlag[g_cartNum,0,2];
//cart stand column error flag
m_safetyCheckData.m_cartStandColumnErr := m_SafetyCheck.m_jntErrFlag[g_cartNum,5,2] OR m_SafetyCheck.m_jntErrFlag[g_cartNum,5,3] OR m_SafetyCheck.m_jntErrFlag[g_cartNum,0,2];
//cart adjust joint contains 6, 7, and 8 joints
m_safetyCheckData.m_cartAdjustErr := m_SafetyCheck.m_jntErrFlag[g_cartNum,6,2] OR m_SafetyCheck.m_jntErrFlag[g_cartNum,6,3] 
															OR m_SafetyCheck.m_jntErrFlag[g_cartNum,7,2] OR m_SafetyCheck.m_jntErrFlag[g_cartNum,7,3]
															OR m_SafetyCheck.m_jntErrFlag[g_cartNum,8,2] OR m_SafetyCheck.m_jntErrFlag[g_cartNum,8,3] OR m_SafetyCheck.m_jntErrFlag[g_cartNum,0,2];
//cart overhang error flag
m_safetyCheckData.m_cartOverhangErr := m_SafetyCheck.m_jntErrFlag[g_cartNum,8,2] OR m_SafetyCheck.m_jntErrFlag[g_cartNum,8,3] OR m_SafetyCheck.m_jntErrFlag[g_cartNum,0,2] OR NOT m_emergencyStopButton;
END_METHOD

METHOD robotPromptMassageCast : BOOL
VAR_IN_OUT CONSTANT
END_VAR

VAR
	i : UDINT;
	m_uiCtrlAdjustFlag : BOOL;
	m_uiCtrlJoystickEnable : BOOL;
	instrument: INT;
END_VAR
FOR i := 1 TO 4 DO
	//0*1021
	m_armsRS[i,1](SET:= m_slaveStatus.m_panelClampErrId[i]=1, 
							RESET1:= NOT m_slaveStatus.m_panelInstallStatus[i], 
							Q1=> m_checkVariable[i].m_promptStatus[1]);
	m_checkVariable[i].m_promptLocation[1] := i + 3;
							
	//0*1022		
	m_armsRS[i,2](SET:= m_slaveStatus.m_panelClampErrId[i]=2, 
							RESET1:= NOT m_slaveStatus.m_panelInstallStatus[i], 
							Q1=> m_checkVariable[i].m_promptStatus[2]);
	m_checkVariable[i].m_promptLocation[2] := i + 3;
	
	//0*1023				
	m_armsRS[i,3](SET:= m_slaveStatus.m_instruReadErrId[i]=1, 
							RESET1:= NOT m_armsRS[i,3].SET OR NOT m_slaveStatus.m_instruInstallStatus[i] , 
							Q1=> m_checkVariable[i].m_promptStatus[3]);
	m_checkVariable[i].m_promptLocation[3] := i + 3;
						
	//0*1024	
	m_armsRS[i,4](SET:= m_slaveStatus.m_instruReadErrId[i]=2, 
							RESET1:=NOT m_armsRS[i,4].SET OR NOT m_slaveStatus.m_instruInstallStatus[i], 
							Q1=> m_checkVariable[i].m_promptStatus[4]);
	m_checkVariable[i].m_promptLocation[4] := i + 3;
	
	//0*1025
	m_armsRS[i,5](SET:= m_slaveStatus.m_instruClampErrId[i]=1, 
							RESET1:=NOT m_armsRS[i,5].SET OR NOT m_slaveStatus.m_instruInstallStatus[i], 
							Q1=> m_checkVariable[i].m_promptStatus[5]);
	m_checkVariable[i].m_promptLocation[5] := i + 3;
	
	 //0*1026
	m_armsRS[i,6](SET:= m_slaveStatus.m_instruClampErrId[i]=2, 
							RESET1:=NOT m_armsRS[i,6].SET OR NOT m_slaveStatus.m_instruInstallStatus[i], 
							Q1=> m_checkVariable[i].m_promptStatus[6]);
	m_checkVariable[i].m_promptLocation[6] := i + 3;
	
	//0*1027
	m_armsRS[i,7](SET:= m_slaveStatus.m_instruReadErrId[i]=3, 
							RESET1:=NOT m_armsRS[i,7].SET OR NOT m_slaveStatus.m_instruInstallStatus[i], 
							Q1=> m_checkVariable[i].m_promptStatus[7]);
	m_checkVariable[i].m_promptLocation[7] := i + 3;
	
	//0*1028	
	m_armsRS[i,8](SET:=NOT m_slaveStatus.m_selfCheckPass[i] AND m_slaveStatus.m_panelInstallStatus[i], 
							RESET1:= NOT m_armsRS[i,8].SET, 
							Q1=> m_checkVariable[i].m_promptStatus[8]);
	m_checkVariable[i].m_promptLocation[8] := i + 3;
				
	//0*1029
	
	 //0*102A
	//m_armsRS[i,10](SET:= m_slaveStatus.m_instruInstallStatus[i] AND NOT m_slaveStatus.m_trocarOnFlag[i], 
	//						RESET1:= NOT m_armsRS[i,10].SET, 
	//						Q1=> m_checkVariable[i].m_promptStatus[10]);
	//m_checkVariable[i].m_promptLocation[10] := i + 3;	
	
	 //0*102B
	FOR j:=1 TO g_mArmNum DO 
		IF i = m_masterRobotData.m_teleSlaveArmIdx[j] THEN
			m_armsRS[i,11](SET:=m_slaveStatus.m_armState[i] = SlaveArmState_Disable AND m_masterRobotData.m_tryMSControl[j] =1, 
									RESET1:= NOT m_armsRS[i,11].SET, 
									Q1=> m_checkVariable[i].m_promptStatus[11]);
			m_checkVariable[i].m_promptLocation[11] := i + 3;
		END_IF
	END_FOR
	
	//0*102C
	FOR j:=1 TO g_mArmNum DO 
		IF i = m_masterRobotData.m_teleSlaveArmIdx[j] THEN
			m_armsRS[i,12](SET:=NOT (SlaveArmState_InstruReady<= m_slaveStatus.m_armState[i] AND m_slaveStatus.m_armState[i] <= SlaveArmState_EndoScope) AND m_masterRobotData.m_tryMSControl[j] =1 AND m_slaveStatus.m_instruStauts[i].m_ready AND m_slaveStatus.m_armState[i] <> SlaveArmState_Disable, 
									RESET1:= NOT m_armsRS[i,12].SET, 
									Q1=> m_checkVariable[i].m_promptStatus[12]);
			m_checkVariable[i].m_promptLocation[12] := i + 3;
		END_IF
	END_FOR
	
				
	//0*102D
	m_armsRS[i,13](SET:= norm(m_slaveStatus.m_masterSlavePoseError[i]) > g_smallNum AND m_slaveStatus.m_armState[i] = SlaveArmState_MasterSlave, 
							RESET1:= NOT m_armsRS[i,13].SET, 
							Q1=> m_checkVariable[i].m_promptStatus[13]);
	m_checkVariable[i].m_promptLocation[13] := i + 3;
	
	
	//0*102E
	m_armsRS[i,14](SET:= NOT SlaveArmControl.m_slaveRobot.m_panelMountedFlag[i] AND (m_masterRobotData.m_tryMSControl[1] =1 OR m_masterRobotData.m_tryMSControl[2] =1) AND m_slaveStatus.m_selfCheckPass[i],
							RESET1:= NOT m_armsRS[i,14].SET, 
							Q1=> m_checkVariable[i].m_promptStatus[14]);
	m_checkVariable[i].m_promptLocation[14] := i + 3;		
	
	//0*102F
	IF InstruType_endoscope = m_slaveStatus.m_instruStauts[i].m_type AND m_slaveStatus.m_endoscopeMounted THEN
		m_scopeArmNoReady := m_slaveStatus.m_armState[i] <> SlaveArmState_ScopeReady AND m_slaveStatus.m_armState[i] <> SlaveArmState_EndoScope;
		m_armsRS[i,15](SET:= (NOT m_slaveStatus.m_endoscopeMounted OR m_scopeArmNoReady) AND (m_masterRobotData.m_tryMSControl[1] =1 OR m_masterRobotData.m_tryMSControl[2] =1), 
								RESET1:= NOT m_armsRS[i,15].SET, 
								Q1=> m_checkVariable[i].m_promptStatus[15]);
		m_checkVariable[i].m_promptLocation[15] := i + 3;	
	ELSE
		m_checkVariable[i].m_promptStatus[15] := FALSE;
	END_IF
END_FOR

//0*102F		预留  没有卡接内窥镜时的检测	
//m_cartRS[15](SET:= NOT m_slaveStatus.m_endoscopeMounted AND (m_masterStatus.m_tryMSControl[1] =1 OR m_masterStatus.m_tryMSControl[2] =1), 
//						RESET1:= NOT m_cartRS[15].SET, 
//						Q1=> m_checkVariable[g_cartNum].m_promptStatus[15]);
//m_checkVariable[g_cartNum].m_promptLocation[15] := 16#0C;


//0*1030			
m_cartRS[16](SET:= NOT m_slaveStatus.m_masterOnLine, 
						RESET1:= m_slaveStatus.m_masterOnLine, 
						Q1=> m_checkVariable[g_cartNum].m_promptStatus[16]);
m_checkVariable[g_cartNum].m_promptLocation[16] := 16#0C;

//0*1031
m_cartRS[17](SET:=m_cartStatus.m_cartDumpEnergy <= 30 , 
						RESET1:= m_cartStatus.m_cartDumpEnergy>30, 
						Q1=> m_checkVariable[g_cartNum].m_promptStatus[17]);
m_checkVariable[g_cartNum].m_promptLocation[17] := g_cartNum + 3;

//0*1032	

//0*1033
m_cartRS[19](SET:= m_cartStatus.m_sdrivingLeverSensorManualFlag, 
						RESET1:=NOT m_cartStatus.m_sdrivingLeverSensorManualFlag, 
						Q1=> m_checkVariable[g_cartNum].m_promptStatus[19]);
m_checkVariable[g_cartNum].m_promptLocation[19] := g_cartNum + 3;

 //0*1034
m_uiCtrlJoystickEnable := m_cartStatus.m_uiControl.m_cameraJoystickEnable OR m_cartStatus.m_uiControl.m_joystickEnable;
m_joysticksTrigger :=  joystickAdjust(m_cartStatus.m_joystickValue);
m_cartRS[20](SET:= m_cartStatus.m_trocarOnFlag=0 AND NOT m_uiCtrlJoystickEnable AND m_joysticksTrigger, 
						RESET1:= NOT m_cartRS[20].SET, 
						Q1=> m_checkVariable[g_cartNum].m_promptStatus[20]);
m_checkVariable[g_cartNum].m_promptLocation[20] := g_cartNum + 3;
					
//0*1035
m_uiCtrlAdjustFlag := m_cartStatus.m_uiControl.m_cameraJoystickEnable OR m_cartStatus.m_uiControl.m_dockingEnable OR m_cartStatus.m_uiControl.m_drapingEnable
							OR m_cartStatus.m_uiControl.m_joystickEnable OR m_cartStatus.m_uiControl.m_packageEnable;
m_cartRS[21](SET:= m_cartStatus.m_trocarOnFlag>0 AND m_uiCtrlAdjustFlag, 
						RESET1:= m_cartStatus.m_trocarOnFlag=0 OR NOT m_uiCtrlAdjustFlag, 
						Q1=> m_checkVariable[g_cartNum].m_promptStatus[21]);
m_checkVariable[g_cartNum].m_promptLocation[21] := g_cartNum + 3;

//0*1036
m_cartRS[22](SET:= m_cartStatus.m_uiControl.m_joystickEnable AND (m_cartStatus.m_jntPosReachLimit[5] OR m_cartStatus.m_jntPosReachLimit[6] OR m_cartStatus.m_jntPosReachLimit[7] OR m_cartStatus.m_jntPosReachLimit[8]), 
						RESET1:= NOT m_cartRS[22].SET, 
						Q1=> m_checkVariable[g_cartNum].m_promptStatus[22]);
m_checkVariable[g_cartNum].m_promptLocation[22] := g_cartNum + 3;
END_METHOD

METHOD warningTone : vec4b
VAR_INPUT
END_VAR
IF (GVL_interactUI.g_curErrType=3) THEN
	warningTone[1] := TRUE;
	warningTone[2] := FALSE;
	warningTone[3] := FALSE;
ELSIF (GVL_interactUI.g_curErrType=2) THEN
	warningTone[1] := FALSE;
	warningTone[2] := TRUE;
	warningTone[3] := FALSE;
//ELSIF (GVL_interactUI.g_curErrType=1) THEN
//	warningTone[1] := TRUE;
//	warningTone[2] := TRUE;
//	warningTone[3] := FALSE;
ELSIF (CartControl.m_cartRobot.m_slaveCart.m_columnJntVel <> 0 AND NOT CartControl.m_cartRobot.m_slaveCart.m_columnAdjustEnable) THEN
	warningTone[1] := FALSE;
	warningTone[2] := FALSE;
	warningTone[3] := TRUE;
//ELSIF m_cartStatus.m_CartState >= CartJointState_HangAdjust AND  m_cartStatus.m_CartState <= CartJointState_StandColuAdjust THEN
//	warningTone[1] := TRUE;
//	warningTone[2] := FALSE;
//	warningTone[3] := TRUE;
ELSE
	warningTone[1] := FALSE;
	warningTone[2] := FALSE;
	warningTone[3] := FALSE;
END_IF
END_METHOD

END_PROGRAM

// ---- SafetyCheck/Fb_SafetyCheck.TcPOU
FUNCTION_BLOCK Fb_SafetyCheck
VAR_INPUT
END_VAR
VAR_OUTPUT
END_VAR
VAR
	i, j:INT;
	m_checkDelay :ARRAY[1..g_maxNum] OF checkDelay;
	m_checkDelayTime :checkDelayTime;
	m_checkPermit:ARRAY[1..g_maxNum] OF  checkPermit;
	
	m_jntErrFlag:ARRAY[1..g_maxNum,0..g_maxArmJoint,1..3] OF BOOL;
	m_armErrFlag:ARRAY [1..g_maxNum,1..3] OF BOOL;
	m_errCode:UDINT;
	
	
	m_errNumType: ARRAY [1..3] OF INT;
	m_ArrayErrCodeType:ARRAY [1..3] OF ARRAY [0..30] OF UDINT;
	m_ArrayErrCodeTypeTest:ARRAY [1..3] OF ARRAY [0..100] OF UDINT;
	m_armErrCodePopup : ARRAY [1..4] OF ARRAY [0..2] OF UDINT;
	m_armErrCodeRefresh : ARRAY [1..4] OF UINT;
	
	//The fault is sent to the UI at the frequency of 0.1S
	m_errCodeUpdateFlag: ARRAY [1..3] OF BOOL;
	m_errCodeUpdateTon: ARRAY [1..3] OF TON;
	
	m_curJntTorqueIOlast :ARRAY [1..g_maxArmNum] OF vec13di;  
	m_cmdJntPosLast : ARRAY [1..g_maxArmNum] OF vec13d;  
	m_cartCurJntTorqueIOlast :vec8di;  
	m_cartCmdJntPosLast : vec8d;  
	o_ErrCode:ARRAY [1..3] OF UDINT;
		
	m_PromptMassBusy:BOOL;
	m_PromptFlag:ARRAY[1..g_maxNum,1..30] OF UINT;
	m_deleteCode:UDINT;
	
	//joint control error
	m_followErrLimit:vec13d:=[g_largeNum, g_largeNum, 0.010, 4(5*g_deg2Rad), 0.010, 5(170*g_deg2Rad)];
END_VAR


VAR CONSTANT
	m_codeUpdateDelay:TIME:=T#0.1S;
	
	//Fault level: 1 indicates  prompt message, 2 indicates a recoverable fault and 3 indicates an unrecoverable fault
	m_promptMessageLevel : UINT :=1;
	m_rcvLevel : UINT:=2;
	m_unrcvLevel : UINT :=3;
END_VAR

METHOD arrayDeleteFrist : ARRAY [0..30] OF UDINT;
VAR_INPUT
	i_array:ARRAY [0..30] OF UDINT;
END_VAR

VAR
	k:INT;
END_VAR

arrayDeleteFrist[30]:=0;

FOR k:=0 TO 29 BY 1 DO
	arrayDeleteFrist[k]:=i_array[k+1];
END_FOR
END_METHOD

METHOD arrayFILO : ARRAY [0..100] OF  UDINT
VAR_INPUT
	i_array:ARRAY[0..100] OF UDINT;
	i_newData:UDINT;
END_VAR

VAR
	i:INT;
END_VAR

FOR i:=0 TO 20 BY 1 DO
	arrayFILO[i]:=i_array[i];
	IF i_array[i]=0 THEN
		arrayFILO[i]:=i_newData;
		EXIT;
	END_IF
END_FOR
END_METHOD

METHOD cartSafetyCheck : BOOL
VAR_INPUT
	i_armId:UDINT;
	i_safetyCheckVar : checkInputVariable;
	i_cartJointData : ST_CartJointData;
END_VAR


VAR
	k:INT;
END_VAR


//驱动器状态监测、驱动器未连接
FOR i:=1 TO g_maxCartJoint BY 1 DO
	m_checkDelay[i_ArmId].T_cartJntStatusErr[i](IN:= (i_safetyCheckVar.m_cartDriverInput[i].m_statusWord=0 AND m_checkPermit[i_ArmId].m_cartJntStatus[i]), PT:=m_checkDelayTime.Ti_CarJntStatus , Q=> , ET=> );
	IF m_checkDelay[i_ArmId].T_cartJntStatusErr[i].Q THEN
		errCodeAssign(i_ArmId, i_ArmId+3,  0, i, 16#3002 ,m_unrcvLevel );
	END_IF
END_FOR



//关节编码器监测
FOR i:=1 TO g_maxCartJoint BY 1 DO
	m_checkDelay[i_ArmId].T_cartLinkEncErr[i](IN:= (i_safetyCheckVar.m_cartDriverInput[i].m_linkEncoder=g_cartMaxLinkEnc[i] OR i_safetyCheckVar.m_cartDriverInput[i].m_linkEncoder=g_cartMinLinkEnc[i]) AND m_checkPermit[i_ArmId].m_cartJntEncErr[i], PT:=m_checkDelayTime.Ti_CarActSec , Q=> , ET=> );
	IF m_checkDelay[i_ArmId].T_cartLinkEncErr[i].Q THEN
		errCodeAssign(i_ArmId, i_ArmId+3,  0, i, 16#3003 ,m_unrcvLevel );
	END_IF
END_FOR


//驱动器错误检测
FOR i:=1 TO g_maxCartJoint BY 1 DO
	m_checkDelay[i_ArmId].T_cartDriveErr[i](IN:= (i_safetyCheckVar.m_cartDriverInput[i].m_driverError AND 16#20)=32 AND m_checkPermit[i_ArmId].m_cartDriveErr[i] , PT:=m_checkDelayTime.Ti_CarDriveErr , Q=> , ET=> );
	IF m_checkDelay[i_ArmId].T_cartDriveErr[i].Q THEN
		errCodeAssign(i_ArmId, i_ArmId+3,  0, i, 16#3004 ,m_unrcvLevel );
	END_IF
END_FOR



//台车双编码器偏差过大
FOR i:=1 TO g_maxCartJoint BY 1 DO
	m_checkDelay[i_ArmId].T_cartJntEncErr[i](IN:= ABS (i_cartJointData.m_curLinkPos[i]-i_cartJointData.m_curJntPos[i])>g_cartMaxJntEncErr[i] AND m_checkPermit[i_ArmId].m_cartJntEncErr[i], PT:=m_checkDelayTime.Ti_CarDualEncDev , Q=> , ET=> );
	IF m_checkDelay[i_ArmId].T_cartJntEncErr[i].Q THEN
		errCodeAssign(i_ArmId, i_ArmId+3,  0, i, 16#3005 ,m_unrcvLevel );
	END_IF
END_FOR


//关节运动超限位
FOR i:=1 TO g_maxCartJoint BY 1 DO
	m_checkDelay[i_ArmId].T_cartOutOfLimit[i](IN:= (i_cartJointData.m_curJntPos[i]>=g_cartMaxJntPos[i] OR i_cartJointData.m_curJntPos[i]<=g_cartMinJntPos[i]) AND m_checkPermit[i_ArmId].m_cartOutOfLimit[i] , PT:=m_checkDelayTime.Ti_CaroutofLimit , Q=> , ET=> );
	IF m_checkDelay[i_ArmId].T_cartOutOfLimit[i].Q THEN
		errCodeAssign(i_ArmId, i_ArmId+3,  0, i, 16#3006 ,m_unrcvLevel );
	END_IF
END_FOR


//驱动器内部通讯错误
FOR i:=1 TO g_maxCartJoint BY 1 DO
	m_checkDelay[i_ArmId].T_cartCurrentIsNotUpdate[i](IN:= (i_safetyCheckVar.m_cartDriverInput[i].m_current=m_cartCurJntTorqueIOlast[i] AND m_checkPermit[i_ArmId].m_cartCurrentIsNotUpdate[i]), PT:=m_checkDelayTime.Ti_CarTorMotor , Q=> , ET=> );
	IF m_checkDelay[i_ArmId].T_cartCurrentIsNotUpdate[i].Q THEN
		errCodeAssign(i_ArmId, i_ArmId+3,  0, i, 16#3009 ,m_unrcvLevel );
	END_IF
	m_cartCurJntTorqueIOlast[i]:=i_safetyCheckVar.m_cartDriverInput[i].m_current;
END_FOR


//关节跟随误差过大
FOR i:=1 TO g_maxCartJoint BY 1 DO
	m_checkDelay[i_ArmId].T_cartJntFollowErr[i](IN:= ABS(i_cartJointData.m_cmdJntPos[i]- i_cartJointData.m_curJntPos[i])>g_cartMaxJntFollowErr[i]  AND m_checkPermit[i_ArmId].m_cartFollowErr[i], PT:=m_checkDelayTime.Ti_CarFollowDev , Q=> , ET=> );
	IF m_checkDelay[i_ArmId].T_cartJntFollowErr[i].Q THEN
		errCodeAssign(i_ArmId, i_ArmId+3,  0, i, 16#2002 ,m_rcvLevel );
	END_IF
END_FOR


//关节速度监控
FOR i:=1 TO g_maxCartJoint BY 1 DO
	m_checkDelay[i_ArmId].T_cartJntVelErr[i](IN:= ABS(i_cartJointData.m_curJntVel[i])>g_cartMaxJntVel[i] AND m_checkPermit[i_ArmId].m_cartJntVelErr[i], PT:=m_checkDelayTime.Ti_CarJntVel , Q=> , ET=> );
	IF m_checkDelay[i_ArmId].T_cartJntVelErr[i].Q THEN
		errCodeAssign(i_ArmId, i_ArmId+3,  0, i, 16#2003 ,m_rcvLevel );
	END_IF
END_FOR


//电流超限监测
FOR i:=1 TO g_maxCartJoint BY 1 DO
	m_checkDelay[i_ArmId].T_cartJntCurrentErr[i](IN:= ABS(i_cartJointData.m_curJntTrq[i])>g_cartMaxJntCurrent[i] AND m_checkPermit[i_ArmId].m_cartJntCurrentErr[i], PT:=m_checkDelayTime.Ti_CarJntCurrent , Q=> , ET=> );
	IF m_checkDelay[i_ArmId].T_cartJntCurrentErr[i].Q THEN
		errCodeAssign(i_ArmId, i_ArmId+3,  0, i, 16#2005 ,m_rcvLevel );
	END_IF
END_FOR


//Ethercat通讯检测
FOR i:=1 TO g_maxCartJoint BY 1 DO
	IF NOT i_safetyCheckVar.m_cartEtherCATState[i].EtherCATState THEN
		errCodeAssign(i_ArmId, i_ArmId+3,  0, i, 16#2006 ,m_rcvLevel );
	END_IF
END_FOR


//鸣志驱动器错误检测
FOR i:=1 TO g_maxCartJoint BY 1 DO
	m_checkDelay[i_ArmId].T_CarMingzhiDriveErr[i](IN:= (i_safetyCheckVar.m_cartDriverInput[i].m_statusWord AND 16#0F)=15  AND m_checkPermit[i_ArmId].m_cartMZDriveErr[i] , PT:=m_checkDelayTime.Ti_CarMZDriveErr , Q=> , ET=> );
	IF m_checkDelay[i_ArmId].T_CarMingzhiDriveErr[i].Q THEN
		errCodeAssign(i_ArmId, i_ArmId+3,  0, i, 16#2009 ,m_rcvLevel );
	END_IF
END_FOR
END_METHOD

PROPERTY checkPermit : REFERENCE TO ARRAY[1..g_maxNum] OF  checkPermit
GET
checkPermit ref= m_checkPermit;
END_GET
SET
END_SET
END_PROPERTY

METHOD electriAngleDev : DINT
VAR_INPUT
	i_motorElectriAngleDev : DINT;
END_VAR

IF i_motorElectriAngleDev > 50000 THEN
	electriAngleDev := i_motorElectriAngleDev - 65535;
ELSIF i_motorElectriAngleDev < -50000 THEN
	electriAngleDev := i_motorElectriAngleDev + 65535;
ELSE
	electriAngleDev := i_motorElectriAngleDev;
END_IF
END_METHOD

METHOD errCodeAssign : BOOL
VAR_INPUT
	i_armId:UDINT;
	i_errLocation:UDINT;
	i_errCodeMode:UDINT;
	i_errJoint:UDINT;
	i_errID:UDINT;
	i_errFlagID :UINT;
END_VAR
IF m_jntErrFlag[i_armId,i_errJoint,i_errFlagID]=FALSE THEN
	m_jntErrFlag[i_armId,i_errJoint,i_errFlagID]:=TRUE;
	m_errCode:=SHL(i_errLocation,24)+SHL(i_errCodeMode,20)+SHL(i_errJoint,16)+i_errID;
	
	
	IF i_errID>=16#3000 THEN
		m_errNumType[m_unrcvLevel]:=LIMIT(0,m_errNumType[m_unrcvLevel]+1,100);
		m_arrayErrCodeType[m_unrcvLevel][m_errNumType[m_unrcvLevel]]:=m_errCode;
		g_arrayErrCodeArm[i_armId]:=arrayFILO(i_Array:= g_arrayErrCodeArm[i_ArmId], i_NewData:=m_errCode );
		m_armErrFlag[i_armId,m_unrcvLevel]:=TRUE;
		
	ELSIF i_errID>=16#2000 THEN
		m_errNumType[m_rcvLevel]:=LIMIT(0,m_errNumType[m_rcvLevel]+1,100);
		m_arrayErrCodeType[m_rcvLevel][m_errNumType[m_rcvLevel]]:=m_errCode;
		g_arrayErrCodeArm[i_armId]:=arrayFILO(i_Array:= g_arrayErrCodeArm[i_ArmId], i_NewData:=m_errCode );
		m_armErrFlag[i_armId,m_rcvLevel]:=TRUE;
		
	END_IF
END_IF
END_METHOD

METHOD errCodeUpdating :ARRAY [1..3] OF UDINT;
VAR_INPUT
END_VAR

m_errCodeUpdateTon[m_unrcvLevel](IN:= NOT m_errCodeUpdateFlag[3], PT:=m_codeUpdateDelay , Q=> m_errCodeUpdateFlag[3], ET=> );
IF m_errCodeUpdateFlag[m_unrcvLevel] THEN
	IF m_errNumType[m_unrcvLevel]>=1 THEN
		m_ArrayErrCodeType[m_unrcvLevel]:=ArrayDeleteFrist(i_Array:=m_ArrayErrCodeType[3]) ;
		o_ErrCode[m_unrcvLevel]:=m_ArrayErrCodeType[m_unrcvLevel][0] ;
		m_ArrayErrCodeTypeTest[m_unrcvLevel]:=arrayFILO(i_Array:= m_ArrayErrCodeTypeTest[m_unrcvLevel], i_NewData:=o_ErrCode[m_unrcvLevel] );
		m_errNumType[m_unrcvLevel]:=m_errNumType[m_unrcvLevel]-1;
	END_IF
END_IF


m_errCodeUpdateTon[m_rcvLevel](IN:= NOT m_errCodeUpdateFlag[m_rcvLevel], PT:=m_codeUpdateDelay , Q=> m_errCodeUpdateFlag[2], ET=> );
IF m_errCodeUpdateFlag[m_rcvLevel] THEN
	IF m_errNumType[m_rcvLevel]>=1 THEN
		m_ArrayErrCodeType[m_rcvLevel]:=ArrayDeleteFrist(i_Array:=m_ArrayErrCodeType[2]) ;
		o_ErrCode[m_rcvLevel]:=m_ArrayErrCodeType[m_rcvLevel][0] ;
		m_ArrayErrCodeTypeTest[m_rcvLevel]:=arrayFILO(i_Array:= m_ArrayErrCodeTypeTest[m_rcvLevel], i_NewData:=o_ErrCode[m_rcvLevel] );
		m_errNumType[m_rcvLevel]:=m_errNumType[m_rcvLevel]-1;
	END_IF
END_IF
END_METHOD

METHOD errFlagReset : BOOL
VAR_INPUT
END_VAR

FOR i := 1 TO g_maxNum DO
	FOR j :=0 TO g_maxArmJoint DO
		m_jntErrFlag[i, j, 2]:=FALSE;
	END_FOR
	m_armErrFlag[i, 2]:=FALSE;
END_FOR

o_ErrCode[2]:=0;
END_METHOD

METHOD poseErrCheck : vec6d
VAR_INPUT
	i_cmdPose : ST_Frame;
	i_curPose :ST_Frame;
END_VAR

VAR
	posErr,oriErr:Vec3d;
	matT,rotErr:Mat3d;
	errAngle :LREAL;
	errAxis :Vec3d;
	i : INT;
END_VAR
vecSub(i_cmdPose.m_pos, i_curPose.m_pos,posErr);

matTranspose(i_cmdPose.m_rot, matT);
matMultiply(matT,i_curPose.m_rot, rotErr);
rot2AngAxis(rotErr, angle=>errAngle, axis=>errAxis);
vecMultiNum(errAxis, errAngle,oriErr);

FOR i := 1 TO 6 DO
	IF i <= 3 THEN
		poseErrCheck[i] := posErr[i];
	ELSE
		poseErrCheck[i] := oriErr[i];
	END_IF
END_FOR
END_METHOD

METHOD promptMassCode : BOOL
VAR_INPUT
	i_PromptStatus:BOOL;
	i_ArmId:UDINT;
	i_ErrID:UDINT;
	i_ErrLocation:UDINT;
END_VAR
VAR
	m_errStatus : UDINT := 0;
	//error ID , 0-15 bit
	m_errId : UDINT;
	m_arrayErrCode : ARRAY [0..30] OF UDINT;
	m_armErrCode : ARRAY [0..2] OF UDINT;
END_VAR

m_PromptMassBusy:=TRUE;

//prompt flag set true
IF i_PromptStatus=TRUE AND m_PromptFlag[i_ArmId,i_ErrID]=0 THEN
	m_PromptFlag[i_ArmId,i_ErrID]:=1;
END_IF

//
IF i_ErrLocation <= 7 AND i_ErrLocation >= 4 THEN
	m_errStatus := 16#00FF;
ELSE
	m_errStatus := 0;
END_IF
m_errId := i_errID+16#1020;

//output prompt error code
IF m_PromptFlag[i_ArmId,i_ErrID]=1 THEN
	m_ErrCode:=SHL(i_ErrLocation,24)+SHL(m_errStatus,16)+i_errID+16#1020;
	vecFIFO(m_ArrayErrCodeType[1] , m_ErrCode , m_arrayErrCode );
	m_ArrayErrCodeType[1]:=m_arrayErrCode;
	IF (m_ErrCode AND 16#00FF0000) = 16#00FF0000 THEN
		vecFIFO(m_armErrCodePopup[i_armId] , m_ErrCode , m_armErrCode );
		m_armErrCodePopup[i_armId] := m_armErrCode;
		m_armErrCodeRefresh[i_armId] := 1;
	END_IF
	m_PromptFlag[i_ArmId,i_ErrID]:=2;
END_IF

//clear prompt error code
IF m_PromptFlag[i_ArmId,i_ErrID]=2 AND i_PromptStatus=FALSE THEN
	m_deleteCode:=SHL(i_ErrLocation,24)+SHL(m_errStatus,16)+i_ErrID+16#1020;
	vecDeleteInput(m_ArrayErrCodeType[1] , m_deleteCode , m_arrayErrCode);
	m_ArrayErrCodeType[1] := m_arrayErrCode;
	IF (m_deleteCode AND 16#00FF0000)  = 16#00FF0000 THEN
		vecDeleteInput(m_armErrCodePopup[i_armId] , m_deleteCode , m_armErrCode );
		m_armErrCodePopup[i_armId] := m_armErrCode;
		m_armErrCodeRefresh[i_armId] := 2;
	END_IF
	//ArrayDeleteInput(i_Array:= m_ArrayErrCodeType[1], i_DeleteCode:=m_deleteCode , o_Array=> m_ArrayErrCodeType[1]);
	m_PromptFlag[i_ArmId,i_ErrID]:=0;
END_IF
o_ErrCode[1]:=m_ArrayErrCodeType[1][0];
m_PromptMassBusy:=FALSE;
END_METHOD

METHOD rcpErrCheck : BOOL
VAR_INPUT
	i_cmdPos : Vec3d;
	i_curPos : Vec3d;
END_VAR
VAR_IN_OUT
	r_errCount:INT;
	r_posErr :Vec3d;
END_VAR

VAR
	err:Vec3d;
END_VAR
vecSub(i_cmdPos, i_curPos,err);
r_posErr:=err;

IF  (norm(err)>g_rcpDeviationThres) THEN
	r_errCount:= r_errCount +1;
ELSE 
	r_errCount:=0;
END_IF
rcpErrCheck := r_errCount >= g_faultTriggerCounts;
END_METHOD

METHOD setupSafetyCheck : BOOL
VAR_INPUT
	i_armId:UDINT;
	i_safetyCheckVar :ARRAY[1..g_maxNum] OF checkInputVariable;
	i_setupJointData : ST_SetupJointData;
END_VAR

VAR
	k:INT;
END_VAR


//驱动器状态监测、驱动器未连接
FOR i:=1 TO g_setupJntNum BY 1 DO
	m_checkDelay[i_ArmId].T_jntStatusErr[i](IN:= (i_safetyCheckVar[i_ArmId].m_setupDriverInput[i].m_statusWord=0 AND m_checkPermit[i_ArmId].m_jntStatusErr[i]), PT:=m_checkDelayTime.Ti_jntStatusErr , Q=> , ET=> );
	IF m_checkDelay[i_ArmId].T_jntStatusErr[i].Q THEN
		errCodeAssign(i_ArmId, i_ArmId+3,  0, i, 16#3002 ,m_unrcvLevel );
	END_IF
END_FOR



//关节编码器监测
FOR i:=1 TO g_setupJntNum BY 1 DO
	m_checkDelay[i_ArmId].T_linkEncErr[i](IN:= (i_safetyCheckVar[i_ArmId].m_setupDriverInput[i].m_linkEncoder=g_maxLinkEnc[i] OR i_safetyCheckVar[i_ArmId].m_setupDriverInput[i].m_linkEncoder=g_minLinkEnc[i]) AND m_checkPermit[i_ArmId].m_linkEncErr[i], PT:=m_checkDelayTime.Ti_linkEncErr , Q=> , ET=> );
	IF m_checkDelay[i_ArmId].T_linkEncErr[i].Q THEN
		errCodeAssign(i_ArmId, i_ArmId+3,  0, i,  16#3003 ,m_unrcvLevel );
	END_IF
END_FOR


//驱动器错误检测
FOR i:=1 TO g_setupJntNum BY 1 DO
	m_checkDelay[i_ArmId].T_DriveErr[i](IN:= (i_safetyCheckVar[i_ArmId].m_setupDriverInput[i].m_driverError AND 16#20)=g_driveErrWord AND m_checkPermit[i_ArmId].m_driveErr[i] , PT:=m_checkDelayTime.Ti_driveErr , Q=> , ET=> );
	IF m_checkDelay[i_ArmId].T_DriveErr[i].Q THEN
		errCodeAssign(i_ArmId, i_ArmId+3,  0, i, 16#3004 ,m_unrcvLevel );
	END_IF
END_FOR


//双编码器偏差过大检测
FOR i:=1 TO g_setupJntNum BY 1 DO
	m_checkDelay[i_ArmId].T_armJntEncErr[i](IN:= ABS(i_setupJointData.m_curLinkPos[i_armId][i]-i_setupJointData.m_curJntPos[i_armId][i])>=g_armMaxJntEncErr[i] AND m_checkPermit[i_ArmId].m_armJntEncErr[i], PT:=m_checkDelayTime.Ti_armJntEncErr , Q=> , ET=> );
	IF m_checkDelay[i_ArmId].T_armJntEncErr[i].Q THEN
		errCodeAssign( i_ArmId, i_ArmId+3,  0, i, 16#3005, m_unrcvLevel );
	END_IF
END_FOR


//关节运动超限位
FOR i:=1 TO g_setupJntNum BY 1 DO
	m_checkDelay[i_ArmId].T_outOfLimit[i](IN:= (i_setupJointData.m_curJntPos[i_armId][i]>=(g_maxJntPos[i_armId,i]+g_armJntPosLimitBuffer[i]) OR i_setupJointData.m_curJntPos[i_armId][i]<=(g_minJntPos[i_armId,i]-g_armJntPosLimitBuffer[i])) AND m_checkPermit[i_ArmId].m_outOfLimit[i] , PT:=m_checkDelayTime.Ti_outofLimit , Q=> , ET=> );
	IF m_checkDelay[i_ArmId].T_outOfLimit[i].Q THEN
		errCodeAssign(i_ArmId, i_ArmId+3,  0, i, 16#3006, m_unrcvLevel );
	END_IF
END_FOR


//电机电角度偏差
FOR i:=1 TO g_setupJntNum BY 1 DO
	IF ABS(electriAngleDev(i_safetyCheckVar[i_armId].m_setupDriverInput[i].m_electriAngleDev))> g_motPhieErrLimit  AND m_checkPermit[i_ArmId].m_motPhieErr[i] THEN
		errCodeAssign(i_ArmId, i_ArmId+3,  0, i, 16#3008, m_unrcvLevel );
	END_IF
END_FOR


//驱动器内部通讯错误
FOR i:=1 TO g_setupJntNum BY 1 DO
	m_checkDelay[i_ArmId].T_currentIsNotUpdate[i](IN:= (i_safetyCheckVar[i_ArmId].m_setupDriverInput[i].m_current=m_curJntTorqueIOlast[i_ArmId][i] AND m_checkPermit[i_ArmId].m_currentIsNotUpdate[i]), PT:=m_checkDelayTime.Ti_currentIsNotUpdate , Q=> , ET=> );
	IF  m_checkDelay[i_ArmId].T_currentIsNotUpdate[i].Q THEN
		errCodeAssign(i_ArmId, i_ArmId+3,  0, i, 16#3009 ,m_unrcvLevel );
	END_IF
	m_curJntTorqueIOlast[i_ArmId][i]:=i_safetyCheckVar[i_ArmId].m_setupDriverInput[i].m_current;
END_FOR


//关节跟随误差过大
FOR i:=1 TO g_setupJntNum BY 1 DO
	m_checkDelay[i_ArmId].T_armJntFollowErr[i](IN:= ABS(i_setupJointData.m_cmdJntPos[i_armId][i]- i_setupJointData.m_curJntPos[i_armId][i])>g_armMaxJntFollowErr[i]  AND m_checkPermit[i_ArmId].m_armJntFollowErr[i], PT:=m_checkDelayTime.Ti_armJntFollowErr , Q=> , ET=> );
	IF m_checkDelay[i_ArmId].T_armJntFollowErr[i].Q THEN
		errCodeAssign(i_ArmId, i_ArmId+3,  0, i, 16#2002, m_rcvLevel );
	END_IF
END_FOR


//关节速度监控
FOR i:=1 TO g_setupJntNum BY 1 DO
	m_checkDelay[i_ArmId].T_jntVelErr[i](IN:= ABS (i_setupJointData.m_curJntVel[i_armId][i])>g_safetyJntVel[i] AND m_checkPermit[i_ArmId].m_jntVelErr[i], PT:=m_checkDelayTime.Ti_jntVelErr , Q=> , ET=> );
	IF m_checkDelay[i_ArmId].T_jntVelErr[i].Q THEN
		errCodeAssign(i_ArmId, i_ArmId+3,  0, i, 16#2003, m_rcvLevel );
	END_IF
END_FOR



//电流超限监测
FOR i:=1 TO g_setupJntNum BY 1 DO
	m_checkDelay[i_ArmId].T_jntCurrentErr[i](IN:= ABS(i_setupJointData.m_rawJntCurrent[i_armId][i])>g_maxJntCurrent[i] AND m_checkPermit[i_ArmId].m_jntCurrentErr[i], PT:=m_checkDelayTime.Ti_jntCurrentErr , Q=> , ET=> );
	IF m_checkDelay[i_ArmId].T_jntCurrentErr[i].Q THEN
		errCodeAssign(i_ArmId, i_ArmId+3,  0, i, 16#2005, m_rcvLevel );
	END_IF
END_FOR


//Ethercat通讯检测
FOR i:=1 TO g_setupJntNum BY 1 DO
	IF NOT i_safetyCheckVar[i_ArmId].m_EtherCATState[i].EtherCATState THEN
		errCodeAssign(i_ArmId, i_ArmId+3, 0, i, 16#2006, m_rcvLevel );
	END_IF
END_FOR


//不动点发生变化监控
m_checkDelay[i_ArmId].T_FixedPointErr(IN:=  i_safetyCheckVar[i_ArmId].m_rcpCheck AND m_checkPermit[i_ArmId].m_fixedPointErr, PT:=m_checkDelayTime.Ti_FixedPointErr , Q=> , ET=> );
IF m_checkDelay[i_ArmId].T_FixedPointErr.Q THEN
	errCodeAssign(i_ArmId, i_ArmId+3,  0, 0, 16#2007, m_rcvLevel );
END_IF


//目标位置指令突变检测
FOR i:=1 TO g_setupJntNum BY 1 DO
	IF (i_setupJointData.m_cmdJntPos[i_armId][i]-m_cmdJntPosLast[i_ArmId][i])>g_maxJntCmdSalta[i] AND m_checkPermit[i_ArmId].m_cmdJntSaltation[i] THEN
		errCodeAssign(i_armId, i_ArmId+3, 0, i, 16#2008, m_rcvLevel );
	END_IF
	m_cmdJntPosLast[i_armId][i] := i_setupJointData.m_cmdJntPos[i_armId][i];
END_FOR


//Deviation between command current and feedback current
FOR i:=1 TO g_setupJntNum BY 1 DO
	IF ABS(i_safetyCheckVar[i_armId].m_slaveDriverOutput[i].m_cmdCurrent-i_safetyCheckVar[i_armId].m_slaveDriverInput[i].m_current)> g_jntCurrentCtrlLimit[i]  AND m_checkPermit[i_armId].m_jntCurrentCtrlErr[i] THEN
		errCodeAssign(i_armId, i_armId+3, 0, i, 16#200B, m_rcvLevel );
	END_IF
END_FOR


//motor encoder mutation detection
FOR i:=1 TO g_setupJntNum BY 1 DO
	IF (i_safetyCheckVar[i_armId].m_motorEncoderSaltaValue[i])>g_maxJntCurSalta[i] THEN
		errCodeAssign(i_armId, i_ArmId+3, 0, i, 16#200C, m_rcvLevel );
	END_IF
END_FOR
END_METHOD

METHOD slaveSafetyCheck : BOOL
VAR_INPUT
	i_armId:UDINT;
	i_safetyCheckVar :ARRAY[1..g_maxNum] OF checkInputVariable;
	i_slaveJointData : ST_SlaveJointData;
END_VAR
//驱动器状态监测、驱动器未连接
FOR i:=1 TO g_sJntNum BY 1 DO
	m_checkDelay[i_ArmId].T_jntStatusErr[i+g_setupJntNum](IN:= (i_safetyCheckVar[i_ArmId].m_slaveDriverInput[i].m_statusWord=0 AND m_checkPermit[i_ArmId].m_jntStatusErr[i+g_setupJntNum]), PT:=m_checkDelayTime.Ti_jntStatusErr , Q=> , ET=> );
	IF m_checkDelay[i_ArmId].T_jntStatusErr[i+g_setupJntNum].Q  THEN
		errCodeAssign(i_ArmId, i_ArmId+3,  0, i+g_setupJntNum, 16#3002 ,m_unrcvLevel );
	END_IF
END_FOR



//关节编码器监测
FOR i:=1 TO g_sJntNum BY 1 DO
	m_checkDelay[i_ArmId].T_linkEncErr[i+g_setupJntNum](IN:= (i_safetyCheckVar[i_ArmId].m_slaveDriverInput[i].m_linkEncoder=g_maxLinkEnc[i] OR i_safetyCheckVar[i_ArmId].m_slaveDriverInput[i].m_linkEncoder=g_minLinkEnc[i]) AND m_checkPermit[i_ArmId].m_linkEncErr[i], PT:=m_checkDelayTime.Ti_linkEncErr , Q=> , ET=> );
	IF m_checkDelay[i_ArmId].T_linkEncErr[i+g_setupJntNum].Q THEN
		errCodeAssign(i_ArmId, i_ArmId+3,  0, i+g_setupJntNum,  16#3003 ,m_unrcvLevel );
	END_IF
END_FOR


//驱动器错误检测
FOR i:=1 TO g_sJntNum BY 1 DO
	m_checkDelay[i_ArmId].T_DriveErr[i+g_setupJntNum](IN:= (i_safetyCheckVar[i_ArmId].m_slaveDriverInput[i].m_driverError AND 16#20)=g_driveErrWord AND m_checkPermit[i_ArmId].m_driveErr[i] , PT:=m_checkDelayTime.Ti_driveErr , Q=> , ET=> );
	IF m_checkDelay[i_ArmId].T_DriveErr[i+g_setupJntNum].Q THEN
		errCodeAssign(i_ArmId, i_ArmId+3,  0, i+g_setupJntNum, 16#3004 ,m_unrcvLevel );
	END_IF
END_FOR


//双编码器偏差过大检测
FOR i:=1 TO g_sJntNum-5 BY 1 DO
	m_checkDelay[i_ArmId].T_armJntEncErr[i+g_setupJntNum](IN:= ABS(i_slaveJointData.m_curLinkPos[i_armId][i]-i_slaveJointData.m_curJntPos[i_armId][i])>=g_armMaxJntEncErr[i+g_setupJntNum] AND m_checkPermit[i_ArmId].m_armJntEncErr[i+g_setupJntNum], PT:=m_checkDelayTime.Ti_armJntEncErr , Q=> , ET=> );
	IF m_checkDelay[i_ArmId].T_armJntEncErr[i+g_setupJntNum].Q THEN
		errCodeAssign( i_ArmId, i_ArmId+3,  0, i+g_setupJntNum, 16#3005, m_unrcvLevel );
	END_IF
END_FOR


//关节运动超限位
FOR i:=1 TO g_sJntNum BY 1 DO
	m_checkDelay[i_ArmId].T_outOfLimit[i+g_setupJntNum](IN:= (i_slaveJointData.m_curJntPos[i_armId][i]>=(g_maxJntPos[i_armId,i+g_setupJntNum]+g_armJntPosLimitBuffer[i+g_setupJntNum]) OR i_slaveJointData.m_curJntPos[i_armId][i]<=(g_minJntPos[i_armId,i+g_setupJntNum]-g_armJntPosLimitBuffer[i+g_setupJntNum])) AND m_checkPermit[i_ArmId].m_outOfLimit[i+g_setupJntNum] , PT:=m_checkDelayTime.Ti_outofLimit , Q=> , ET=> );
	IF m_checkDelay[i_ArmId].T_outOfLimit[i+g_setupJntNum].Q THEN
		errCodeAssign(i_ArmId, i_ArmId+3,  0, i+g_setupJntNum, 16#3006, m_unrcvLevel );
	END_IF
END_FOR


//电机电角度偏差
FOR i:=1 TO g_sJntNum BY 1 DO
	IF ABS(electriAngleDev(i_safetyCheckVar[i_armId].m_slaveDriverInput[i].m_electriAngleDev))> g_motPhieErrLimit  AND m_checkPermit[i_ArmId].m_motPhieErr[i+g_setupJntNum] THEN
		errCodeAssign(i_ArmId, i_ArmId+3,  0, i+g_setupJntNum, 16#3008, m_unrcvLevel );
	END_IF
END_FOR


//驱动器内部通讯错误
FOR i:=1 TO g_sJntNum BY 1 DO
	m_checkDelay[i_ArmId].T_currentIsNotUpdate[i+g_setupJntNum](IN:= (i_safetyCheckVar[i_ArmId].m_slaveDriverInput[i].m_current=m_curJntTorqueIOlast[i_ArmId][i+g_setupJntNum] AND m_checkPermit[i_ArmId].m_currentIsNotUpdate[i+g_setupJntNum]), PT:=m_checkDelayTime.Ti_currentIsNotUpdate , Q=> , ET=> );
	IF  m_checkDelay[i_ArmId].T_currentIsNotUpdate[i+g_setupJntNum].Q THEN
		errCodeAssign(i_ArmId, i_ArmId+3,  0, i+g_setupJntNum, 16#3009 ,m_unrcvLevel );
	END_IF
	m_curJntTorqueIOlast[i_ArmId][i+g_setupJntNum]:=i_safetyCheckVar[i_ArmId].m_slaveDriverInput[i].m_current;
END_FOR


//关节跟随误差过大---1028
FOR i:=1 TO g_sJntNum BY 1 DO
	(*
	m_checkDelay[i_ArmId].T_armJntFollowErr[i+g_setupJntNum](IN:= ABS(i_slaveJointData.m_cmdJntPos[i_armId][i]- i_slaveJointData.m_curJntPos[i_armId][i])>g_armMaxJntFollowErr[i+g_setupJntNum]  AND m_checkPermit[i_ArmId].m_armJntFollowErr[i+g_setupJntNum], PT:=m_checkDelayTime.Ti_armJntFollowErr , Q=> , ET=> );
	IF m_checkDelay[i_ArmId].T_armJntFollowErr[i+g_setupJntNum].Q THEN
		errCodeAssign(i_ArmId, i_ArmId+3,  0, i+g_setupJntNum, 16#2002, m_rcvLevel );
	END_IF
	*)
	
	//update the control error limit
	IF (SlaveArmControl.m_slaveRobot.m_stiffChanged[i_ArmId]=TRUE) THEN
		m_followErrLimit:=g_armMaxJntFollowErrSoftStiff;
	ELSE
		m_followErrLimit:=g_armMaxJntFollowErr;
	END_IF
	
	//check
	m_checkDelay[i_ArmId].T_armJntFollowErr[i+g_setupJntNum](IN:= ABS(i_slaveJointData.m_cmdJntPos[i_armId][i]- i_slaveJointData.m_curJntPos[i_armId][i])>m_followErrLimit[i+g_setupJntNum]  AND m_checkPermit[i_ArmId].m_armJntFollowErr[i+g_setupJntNum], PT:=m_checkDelayTime.Ti_armJntFollowErr , Q=> , ET=> );
	IF m_checkDelay[i_ArmId].T_armJntFollowErr[i+g_setupJntNum].Q THEN
		errCodeAssign(i_ArmId, i_ArmId+3,  0, i+g_setupJntNum, 16#2002, m_rcvLevel );
	END_IF	
END_FOR


//关节速度监控
FOR i:=1 TO g_sJntNum-5 BY 1 DO
	m_checkDelay[i_ArmId].T_jntVelErr[i+g_setupJntNum](IN:= ABS (i_slaveJointData.m_curJntVel[i_armId][i])>g_safetyJntVel[i+g_setupJntNum] AND m_checkPermit[i_ArmId].m_jntVelErr[i+g_setupJntNum], PT:=m_checkDelayTime.Ti_jntVelErr , Q=> , ET=> );
	IF m_checkDelay[i_ArmId].T_jntVelErr[i+g_setupJntNum].Q THEN
		errCodeAssign(i_ArmId, i_ArmId+3,  0, i+g_setupJntNum, 16#2003, m_rcvLevel );
	END_IF
END_FOR


// TODO: replaced with cartesin twist check
//笛卡尔空间指令与位置偏差检测
//FOR i:=1 TO 6 BY 1 DO
//	m_checkDelay[i_ArmId].T_spacePoseErr[i](IN:= i_safetyCheckVar[i_ArmId].m_spacePoseErr[i]> g_maxCartPoseErr[i] AND m_checkPermit[i_ArmId].m_spacePoseErr[i], PT:=m_checkDelayTime.Ti_spacePoseErr , Q=> , ET=> );
//	IF m_checkDelay[i_ArmId].T_spacePoseErr[i].Q THEN
//		errCodeAssign(i_ArmId, i_ArmId+3, 1, i, 16#2004, m_rcvLevel );
//	END_IF
//END_FOR


//电流超限监测
FOR i:=1 TO g_sJntNum BY 1 DO
	m_checkDelay[i_ArmId].T_jntCurrentErr[i+g_setupJntNum](IN:= ABS(i_slaveJointData.m_rawJntCurrent[i_armId][i])>g_maxJntCurrent[i+g_setupJntNum] AND m_checkPermit[i_ArmId].m_jntCurrentErr[i+g_setupJntNum], PT:=m_checkDelayTime.Ti_jntCurrentErr , Q=> , ET=> );
	IF m_checkDelay[i_ArmId].T_jntCurrentErr[i+g_setupJntNum].Q THEN
		errCodeAssign(i_ArmId, i_ArmId+3,  0, i+g_setupJntNum, 16#2005, m_rcvLevel );
	END_IF
END_FOR


//Ethercat通讯检测
FOR i:=1 TO g_sJntNum BY 1 DO
	IF NOT i_safetyCheckVar[i_ArmId].m_EtherCATState[i+g_setupJntNum].EtherCATState THEN
		errCodeAssign(i_ArmId, i_ArmId+3, 0, i+g_setupJntNum, 16#2006, m_rcvLevel );
	END_IF
END_FOR


//目标位置指令突变检测
FOR i:=1 TO g_sJntNum BY 1 DO
	m_checkDelay[i_ArmId].T_jntCmdSalta[i+g_setupJntNum](IN:= m_checkPermit[i_ArmId].m_cmdJntSaltation[i+g_setupJntNum], PT:=m_checkDelayTime.Ti_jntCmdSaltationErr , Q=> , ET=> );
	IF m_checkDelay[i_ArmId].T_jntCmdSalta[i+g_setupJntNum].Q THEN
		IF (i_slaveJointData.m_cmdJntPos[i_armId][i]-m_cmdJntPosLast[i_ArmId][i+g_setupJntNum])>g_maxJntCmdSalta[i+g_setupJntNum] THEN
			errCodeAssign(i_ArmId, i_ArmId+3, 0, i+g_setupJntNum, 16#2008, m_rcvLevel );
		END_IF
	END_IF
	m_cmdJntPosLast[i_ArmId][i+g_setupJntNum] := i_slaveJointData.m_cmdJntPos[i_armId][i];
END_FOR


//Deviation between command current and feedback current
//FOR i:=1 TO g_sJntNum BY 1 DO
//	IF ABS(i_safetyCheckVar[i_armId].m_slaveDriverOutput[i].m_cmdCurrent-i_safetyCheckVar[i_armId].m_slaveDriverInput[i].m_current)> g_jntCurrentCtrlLimit[i+g_setupJntNum]  AND m_checkPermit[i_armId].m_jntCurrentCtrlErr[i+g_setupJntNum] THEN
//		errCodeAssign(i_armId, i_armId+3, 0, i+g_setupJntNum, 16#200B, m_rcvLevel );
//	END_IF
//END_FOR


//motor encoder mutation detection
FOR i:=1 TO g_sJntNum BY 1 DO
	IF (i_safetyCheckVar[i_armId].m_motorEncoderSaltaValue[i+g_setupJntNum])>g_maxJntCurSalta[i+g_setupJntNum] THEN
		errCodeAssign(i_armId, i_ArmId+3, 0, i+g_setupJntNum, 16#200C, m_rcvLevel );
	END_IF
END_FOR


//器械张开角度过大或过小
IF (i_safetyCheckVar[i_ArmId].m_instruOpenAngle> g_maxInstruOpen OR i_safetyCheckVar[i_ArmId].m_instruOpenAngle< 0) AND m_checkPermit[i_ArmId].m_instruOpenAngle THEN
	errCodeAssign(i_ArmId, i_ArmId+3, 0, 0, 16#200D, m_rcvLevel );
END_IF
END_METHOD

METHOD systemSafetyCheck : BOOL
VAR_INPUT
	i_armId:UDINT;
	i_safetyCheckVar :ARRAY[1..g_maxNum] OF checkInputVariable;
	i_cartJointData : ST_CartJointData;
	i_setupJointData : ST_SetupJointData;
	i_slaveJointData : ST_SlaveJointData;
END_VAR

VAR
	k:INT;
END_VAR

IF i_armId =g_cartNum THEN 
	//cart safrty check
	cartSafetyCheck(i_armId,i_safetyCheckVar[i_armId],i_cartJointData);
ELSE
	//EmergencyStopButton
	IF NOT i_safetyCheckVar[i_ArmId].EmergencyStop OR m_jntErrFlag[i_armId,0,3] THEN
		errCodeAssign(i_ArmId, 16#0C, 0, 0, 16#3001, m_unrcvLevel);
		RETURN;
	END_IF
	//setup arms safety check
	setupSafetyCheck(i_armId,i_safetyCheckVar,i_setupJointData);
	//slave arms safety check
	slaveSafetyCheck(i_armId,i_safetyCheckVar,i_slaveJointData);
END_IF

//StopButton
IF NOT i_safetyCheckVar[i_ArmId].SlaveStopButton OR i_safetyCheckVar[i_ArmId].PCStopButton=0 OR i_safetyCheckVar[i_ArmId].MasterStopButton THEN
	errCodeAssign(i_ArmId, 16#0C, 0, 0, 16#2001, m_rcvLevel );
END_IF

//prompt message
FOR i:=1 TO 30 BY 1 DO
	PromptMassCode( i_safetyCheckVar[i_ArmId].m_promptStatus[i], i_ArmId,  i,  i_safetyCheckVar[i_ArmId].m_promptLocation[i]);
END_FOR
END_METHOD

METHOD vecDeleteInput : BOOL
VAR_IN_OUT CONSTANT
	vecA :ARRAY[*] OF UDINT;
END_VAR

VAR_INPUT
	i_deleteCode :UDINT;
END_VAR

VAR_IN_OUT
	vecB : ARRAY[*] OF UDINT;
END_VAR

VAR
	m :DINT;
	i :DINT;
	Falg:BOOL;
END_VAR
m:=UPPER_BOUND(vecA,1);

FOR i:=0 TO m BY 1 DO 
	IF vecA[i]=i_DeleteCode THEN
		Falg:=TRUE;
	END_IF
	
	IF Falg=TRUE THEN
		vecB[i]:=vecA[i+1];
	ELSE
		vecB[i]:=vecA[i];
	END_IF
END_FOR
vecB[m]:=0;
END_METHOD

METHOD vecFIFO : BOOL
VAR_IN_OUT CONSTANT
	vecA :ARRAY[*] OF UDINT;
END_VAR

VAR_INPUT
	i_newData :UDINT;
END_VAR

VAR_IN_OUT
	vecB : ARRAY[*] OF UDINT;
END_VAR

VAR
	m :DINT;
	i :DINT;
END_VAR
m:=UPPER_BOUND(vecA,1);

FOR i:=0 TO m DO
	vecB[i+1]:=vecA[i];
END_FOR

vecB[0]:=i_newData;
END_METHOD

END_FUNCTION_BLOCK

// ---- AgiMaths/MatrixLib/rot2AngAxis.TcPOU
FUNCTION rot2AngAxis : bool
VAR_IN_OUT CONSTANT
	rot : Mat3d;
END_VAR
VAR_OUTPUT
	angle: LREAL;
	axis : Vec3d;
END_VAR
VAR
	tmp:LREAL;
END_VAR

tmp:=LIMIT(-1, (rot[1,1]+rot[2,2]+rot[3,3]-1)/2 , 1);
angle := ACOS(tmp);

